LIN {X 0,Y 488.681,Z 523.609,A -85,B 0,C 180,E1 -6353.868,E2 -6353.868} C_VEL
LIN {X 0,Y 488.74,Z 523.606,A -85,B 0,C 180,E1 -6356.877,E2 -6356.877} C_VEL
LIN {X 0,Y 488.729,Z 523.605,A -85,B 0,C 180,E1 -6359.78,E2 -6359.78} C_VEL
LIN {X 0,Y 488.797,Z 523.6,A -85,B 0,C 180,E1 -6363.056,E2 -6363.056} C_VEL
LIN {X 0,Y 488.688,Z 523.606,A -85,B 0,C 180,E1 -6366.254,E2 -6366.254} C_VEL
LIN {X 0,Y 488.769,Z 523.791,A -85,B 0,C 180,E1 -6368.6,E2 -6368.6} C_VEL
LIN {X 0,Y 489.922,Z 530.451,A -85,B 0,C 180,E1 -6370.08,E2 -6370.08} C_VEL
LIN {X 0,Y 489.464,Z 545.093,A -85,B 0,C 180,E1 -6373.096,E2 -6373.096} C_VEL
LIN {X 0,Y 489.361,Z 548.713,A -85,B 0,C 180,E1 -6373.771,E2 -6373.771} C_VEL
LIN {X 0,Y 491.805,Z 562.137,A -85,B 0,C 180,E1 -6374.082,E2 -6374.082} C_VEL
LIN {X 0,Y 491.211,Z 655.586,A -85,B 0,C 180,E1 -6375.473,E2 -6375.473} C_VEL
LIN {X 0,Y 490.919,Z 668.738,A -85,B 0,C 180,E1 -6375.834,E2 -6375.834} C_VEL
LIN {X 0,Y 490.606,Z 680.814,A -85,B 0,C 180,E1 -6376.327,E2 -6376.327} C_VEL
LIN {X 0,Y 490.275,Z 691.758,A -85,B 0,C 180,E1 -6376.924,E2 -6376.924} C_VEL
LIN {X 0,Y 489.93,Z 702.578,A -85,B 0,C 180,E1 -6377.679,E2 -6377.679} C_VEL
LIN {X 0,Y 489.463,Z 713.275,A -85,B 0,C 180,E1 -6378.613,E2 -6378.613} C_VEL
LIN {X 0,Y 489.087,Z 722.892,A -85,B 0,C 180,E1 -6379.652,E2 -6379.652} C_VEL
LIN {X 0,Y 488.737,Z 730.772,A -85,B 0,C 180,E1 -6380.689,E2 -6380.689} C_VEL
LIN {X 0,Y 488.455,Z 738.473,A -85,B 0,C 180,E1 -6381.935,E2 -6381.935} C_VEL
LIN {X 0,Y 488.183,Z 745.539,A -85,B 0,C 180,E1 -6383.386,E2 -6383.386} C_VEL
LIN {X 0,Y 488.073,Z 750.246,A -85,B 0,C 180,E1 -6384.629,E2 -6384.629} C_VEL
LIN {X 0,Y 488.068,Z 753.846,A -85,B 0,C 180,E1 -6385.871,E2 -6385.871} C_VEL
LIN {X 0,Y 487.979,Z 755.709,A -85,B 0,C 180,E1 -6386.697,E2 -6386.697} C_VEL
LIN {X 0,Y 487.933,Z 757.116,A -85,B 0,C 180,E1 -6387.523,E2 -6387.523} C_VEL
LIN {X 0,Y 487.834,Z 758.735,A -85,B 0,C 180,E1 -6389.174,E2 -6389.174} C_VEL
LIN {X 0,Y 487.819,Z 758.973,A -85,B 0,C 180,E1 -6389.999,E2 -6389.999} C_VEL
LIN {X 0,Y 487.834,Z 758.789,A -85,B 0,C 180,E1 -6390.825,E2 -6390.825} C_VEL
LIN {X 0,Y 487.933,Z 757.242,A -85,B 0,C 180,E1 -6392.476,E2 -6392.476} C_VEL
LIN {X 0,Y 487.979,Z 755.889,A -85,B 0,C 180,E1 -6393.302,E2 -6393.302} C_VEL
LIN {X 0,Y 488.012,Z 753.026,A -85,B 0,C 180,E1 -6394.542,E2 -6394.542} C_VEL
LIN {X 0,Y 488.204,Z 748.083,A -85,B 0,C 180,E1 -6396.069,E2 -6396.069} C_VEL
LIN {X 0,Y 488.28,Z 742.168,A -85,B 0,C 180,E1 -6397.442,E2 -6397.442} C_VEL
LIN {X 0,Y 488.598,Z 735.386,A -85,B 0,C 180,E1 -6398.686,E2 -6398.686} C_VEL
LIN {X 0,Y 488.907,Z 726.92,A -85,B 0,C 180,E1 -6399.932,E2 -6399.932} C_VEL
LIN {X 0,Y 489.272,Z 718.209,A -85,B 0,C 180,E1 -6400.971,E2 -6400.971} C_VEL
LIN {X 0,Y 489.748,Z 707.478,A -85,B 0,C 180,E1 -6402.009,E2 -6402.009} C_VEL
LIN {X 0,Y 490.074,Z 696.27,A -85,B 0,C 180,E1 -6402.873,E2 -6402.873} C_VEL
LIN {X 0,Y 490.496,Z 684.645,A -85,B 0,C 180,E1 -6403.569,E2 -6403.569} C_VEL
LIN {X 0,Y 490.899,Z 671.996,A -85,B 0,C 180,E1 -6404.138,E2 -6404.138} C_VEL
LIN {X 0,Y 491.147,Z 659.517,A -85,B 0,C 180,E1 -6404.528,E2 -6404.528} C_VEL
LIN {X 0,Y 491.348,Z 643.583,A -85,B 0,C 180,E1 -6404.813,E2 -6404.813} C_VEL
LIN {X 0,Y 491.714,Z 561.306,A -85,B 0,C 180,E1 -6406.023,E2 -6406.023} C_VEL
LIN {X 0,Y 489.374,Z 548.902,A -85,B 0,C 180,E1 -6406.31,E2 -6406.31} C_VEL
LIN {X 0,Y 489.362,Z 547.534,A -85,B 0,C 180,E1 -6406.498,E2 -6406.498} C_VEL
LIN {X 0,Y 489.893,Z 531.929,A -85,B 0,C 180,E1 -6409.701,E2 -6409.701} C_VEL
LIN {X 0,Y 489.546,Z 527.949,A -85,B 0,C 180,E1 -6410.555,E2 -6410.555} C_VEL
LIN {X 0,Y 488.755,Z 523.632,A -85,B 0,C 180,E1 -6411.565,E2 -6411.565} C_VEL
LIN {X 0,Y 488.746,Z 523.607,A -85,B 0,C 180,E1 -6415.052,E2 -6415.052} C_VEL
LIN {X 0,Y 488.746,Z 523.608,A -85,B 0,C 180,E1 -6417.396,E2 -6417.396} C_VEL
LIN {X 0,Y 488.709,Z 523.603,A -85,B 0,C 180,E1 -6420.362,E2 -6420.362} C_VEL
LIN {X 0,Y 488.734,Z 523.608,A -85,B 0,C 180,E1 -6423.484,E2 -6423.484} C_VEL
LIN {X 0,Y 488.687,Z 523.606,A -85,B 0,C 180,E1 -6426.355,E2 -6426.355} C_VEL
LIN {X 0,Y 488.699,Z 523.611,A -85,B 0,C 180,E1 -6429.253,E2 -6429.253} C_VEL
LIN {X 0,Y 488.721,Z 523.61,A -85,B 0,C 180,E1 -6431.601,E2 -6431.601} C_VEL
LIN {X 0,Y 488.708,Z 523.601,A -85,B 0,C 180,E1 -6434.8,E2 -6434.8} C_VEL
LIN {X 0,Y 488.687,Z 523.616,A -85,B 0,C 180,E1 -6437.474,E2 -6437.474} C_VEL
LIN {X 0,Y 488.744,Z 523.595,A -85,B 0,C 180,E1 -6440.75,E2 -6440.75} C_VEL
LIN {X 0,Y 488.681,Z 523.611,A -85,B 0,C 180,E1 -6443.868,E2 -6443.868} C_VEL
LIN {X 0,Y 488.734,Z 523.603,A -85,B 0,C 180,E1 -6446.877,E2 -6446.877} C_VEL
LIN {X 0,Y 488.728,Z 523.607,A -85,B 0,C 180,E1 -6449.781,E2 -6449.781} C_VEL
LIN {X 0,Y 488.793,Z 523.593,A -85,B 0,C 180,E1 -6453.054,E2 -6453.054} C_VEL
LIN {X 0,Y 488.687,Z 523.606,A -85,B 0,C 180,E1 -6456.254,E2 -6456.254} C_VEL
LIN {X 0,Y 488.739,Z 523.602,A -85,B 0,C 180,E1 -6459.175,E2 -6459.175} C_VEL
LIN {X 0,Y 488.752,Z 523.604,A -85,B 0,C 180,E1 -6461.627,E2 -6461.627} C_VEL
LIN {X 0,Y 488.754,Z 523.597,A -85,B 0,C 180,E1 -6464.999,E2 -6464.999} C_VEL
LIN {X 0,Y 488.798,Z 523.592,A -85,B 0,C 180,E1 -6468.387,E2 -6468.387} C_VEL
LIN {X 0,Y 488.811,Z 523.597,A -85,B 0,C 180,E1 -6471.733,E2 -6471.733} C_VEL
LIN {X 0,Y 488.849,Z 523.588,A -85,B 0,C 180,E1 -6474.224,E2 -6474.224} C_VEL
LIN {X 0,Y 488.954,Z 523.576,A -85,B 0,C 180,E1 -6477.529,E2 -6477.529} C_VEL
LIN {X 0,Y 488.962,Z 523.576,A -85,B 0,C 180,E1 -6480,E2 -6480} C_VEL
LIN {X 0,Y 488.955,Z 523.571,A -85,B 0,C 180,E1 -6482.471,E2 -6482.471} C_VEL
LIN {X 0,Y 488.848,Z 523.593,A -85,B 0,C 180,E1 -6485.776,E2 -6485.776} C_VEL
LIN {X 0,Y 488.81,Z 523.591,A -85,B 0,C 180,E1 -6488.267,E2 -6488.267} C_VEL
LIN {X 0,Y 488.822,Z 523.596,A -85,B 0,C 180,E1 -6491.612,E2 -6491.612} C_VEL
LIN {X 0,Y 488.754,Z 523.599,A -85,B 0,C 180,E1 -6495.001,E2 -6495.001} C_VEL
LIN {X 0,Y 488.747,Z 523.6,A -85,B 0,C 180,E1 -6498.442,E2 -6498.442} C_VEL
LIN {X 0,Y 488.7,Z 523.606,A -85,B 0,C 180,E1 -6501.071,E2 -6501.071} C_VEL
LIN {X 0,Y 488.687,Z 523.615,A -85,B 0,C 180,E1 -6503.746,E2 -6503.746} C_VEL
LIN {X 0,Y 488.792,Z 523.592,A -85,B 0,C 180,E1 -6506.946,E2 -6506.946} C_VEL
LIN {X 0,Y 488.703,Z 523.604,A -85,B 0,C 180,E1 -6510.364,E2 -6510.364} C_VEL
LIN {X 0,Y 488.73,Z 523.609,A -85,B 0,C 180,E1 -6513.485,E2 -6513.485} C_VEL
LIN {X 0,Y 488.683,Z 523.599,A -85,B 0,C 180,E1 -6516.356,E2 -6516.356} C_VEL
LIN {X 0,Y 488.696,Z 523.609,A -85,B 0,C 180,E1 -6519.255,E2 -6519.255} C_VEL
LIN {X 0,Y 488.704,Z 523.609,A -85,B 0,C 180,E1 -6521.601,E2 -6521.601} C_VEL
LIN {X 0,Y 488.707,Z 523.606,A -85,B 0,C 180,E1 -6524.802,E2 -6524.802} C_VEL
LIN {X 0,Y 488.728,Z 523.604,A -85,B 0,C 180,E1 -6527.48,E2 -6527.48} C_VEL
LIN {X 0,Y 488.739,Z 523.598,A -85,B 0,C 180,E1 -6530.751,E2 -6530.751} C_VEL
LIN {X 0,Y 488.681,Z 523.613,A -85,B 0,C 180,E1 -6533.869,E2 -6533.869} C_VEL
LIN {X 0,Y 488.737,Z 523.596,A -85,B 0,C 180,E1 -6536.878,E2 -6536.878} C_VEL
LIN {X 0,Y 488.722,Z 523.579,A -85,B 0,C 180,E1 -6539.782,E2 -6539.782} C_VEL
LIN {X 0,Y 488.791,Z 523.587,A -85,B 0,C 180,E1 -6543.057,E2 -6543.057} C_VEL
LIN {X 0,Y 488.791,Z 523.664,A -85,B 0,C 180,E1 -6544.812,E2 -6544.812} C_VEL
LIN {X 0,Y 489.553,Z 527.685,A -85,B 0,C 180,E1 -6545.624,E2 -6545.624} C_VEL
LIN {X 0,Y 490.749,Z 534.364,A -85,B 0,C 180,E1 -6546.859,E2 -6546.859} C_VEL
LIN {X 0,Y 490.077,Z 551.858,A -85,B 0,C 180,E1 -6549.869,E2 -6549.869} C_VEL
LIN {X 0,Y 489.463,Z 569.569,A -85,B 0,C 180,E1 -6552.882,E2 -6552.882} C_VEL
LIN {X 0,Y 489.365,Z 574.51,A -85,B 0,C 180,E1 -6553.695,E2 -6553.695} C_VEL
LIN {X 0,Y 490.061,Z 579.414,A -85,B 0,C 180,E1 -6553.83,E2 -6553.83} C_VEL
LIN {X 0,Y 491.733,Z 590.249,A -85,B 0,C 180,E1 -6554.047,E2 -6554.047} C_VEL
LIN {X 0,Y 491.141,Z 682.718,A -85,B 0,C 180,E1 -6555.419,E2 -6555.419} C_VEL
LIN {X 0,Y 490.851,Z 695.983,A -85,B 0,C 180,E1 -6555.781,E2 -6555.781} C_VEL
LIN {X 0,Y 490.517,Z 708.151,A -85,B 0,C 180,E1 -6556.273,E2 -6556.273} C_VEL
LIN {X 0,Y 490.094,Z 720.568,A -85,B 0,C 180,E1 -6556.956,E2 -6556.956} C_VEL
LIN {X 0,Y 489.627,Z 732.037,A -85,B 0,C 180,E1 -6557.778,E2 -6557.778} C_VEL
LIN {X 0,Y 489.256,Z 742.483,A -85,B 0,C 180,E1 -6558.714,E2 -6558.714} C_VEL
LIN {X 0,Y 488.874,Z 751.025,A -85,B 0,C 180,E1 -6559.649,E2 -6559.649} C_VEL
LIN {X 0,Y 488.593,Z 758.906,A -85,B 0,C 180,E1 -6560.688,E2 -6560.688} C_VEL
LIN {X 0,Y 488.327,Z 766.606,A -85,B 0,C 180,E1 -6561.934,E2 -6561.934} C_VEL
LIN {X 0,Y 488.1,Z 773.701,A -85,B 0,C 180,E1 -6563.386,E2 -6563.386} C_VEL
LIN {X 0,Y 488.033,Z 778.425,A -85,B 0,C 180,E1 -6564.63,E2 -6564.63} C_VEL
LIN {X 0,Y 487.934,Z 782.035,A -85,B 0,C 180,E1 -6565.871,E2 -6565.871} C_VEL
LIN {X 0,Y 487.965,Z 783.899,A -85,B 0,C 180,E1 -6566.698,E2 -6566.698} C_VEL
LIN {X 0,Y 487.89,Z 786.286,A -85,B 0,C 180,E1 -6568.35,E2 -6568.35} C_VEL
LIN {X 0,Y 487.819,Z 787.107,A -85,B 0,C 180,E1 -6570.001,E2 -6570.001} C_VEL
LIN {X 0,Y 487.89,Z 786.283,A -85,B 0,C 180,E1 -6571.652,E2 -6571.652} C_VEL
LIN {X 0,Y 487.965,Z 783.892,A -85,B 0,C 180,E1 -6573.303,E2 -6573.303} C_VEL
LIN {X 0,Y 487.928,Z 780.957,A -85,B 0,C 180,E1 -6574.544,E2 -6574.544} C_VEL
LIN {X 0,Y 488.06,Z 776.989,A -85,B 0,C 180,E1 -6575.786,E2 -6575.786} C_VEL
LIN {X 0,Y 488.184,Z 770.876,A -85,B 0,C 180,E1 -6577.237,E2 -6577.237} C_VEL
LIN {X 0,Y 488.382,Z 764.198,A -85,B 0,C 180,E1 -6578.483,E2 -6578.483} C_VEL
LIN {X 0,Y 488.702,Z 755.914,A -85,B 0,C 180,E1 -6579.729,E2 -6579.729} C_VEL
LIN {X 0,Y 489.013,Z 747.424,A -85,B 0,C 180,E1 -6580.769,E2 -6580.769} C_VEL
LIN {X 0,Y 489.508,Z 736.936,A -85,B 0,C 180,E1 -6581.806,E2 -6581.806} C_VEL
LIN {X 0,Y 489.842,Z 725.58,A -85,B 0,C 180,E1 -6582.711,E2 -6582.711} C_VEL
LIN {X 0,Y 490.288,Z 713.26,A -85,B 0,C 180,E1 -6583.471,E2 -6583.471} C_VEL
LIN {X 0,Y 490.725,Z 700.919,A -85,B 0,C 180,E1 -6584.039,E2 -6584.039} C_VEL
LIN {X 0,Y 491.05,Z 688.242,A -85,B 0,C 180,E1 -6584.453,E2 -6584.453} C_VEL
LIN {X 0,Y 491.266,Z 675.001,A -85,B 0,C 180,E1 -6584.711,E2 -6584.711} C_VEL
LIN {X 0,Y 491.59,Z 588.729,A -85,B 0,C 180,E1 -6585.98,E2 -6585.98} C_VEL
LIN {X 0,Y 489.357,Z 574.659,A -85,B 0,C 180,E1 -6586.292,E2 -6586.292} C_VEL
LIN {X 0,Y 489.946,Z 556.914,A -85,B 0,C 180,E1 -6589.265,E2 -6589.265} C_VEL
LIN {X 0,Y 490.637,Z 537.874,A -85,B 0,C 180,E1 -6592.531,E2 -6592.531} C_VEL
LIN {X 0,Y 490.755,Z 534.35,A -85,B 0,C 180,E1 -6593.143,E2 -6593.143} C_VEL
LIN {X 0,Y 488.834,Z 523.999,A -85,B 0,C 180,E1 -6595.075,E2 -6595.075} C_VEL
LIN {X 0,Y 488.776,Z 523.603,A -85,B 0,C 180,E1 -6595.263,E2 -6595.263} C_VEL
LIN {X 0,Y 488.75,Z 523.605,A -85,B 0,C 180,E1 -6597.397,E2 -6597.397} C_VEL
LIN {X 0,Y 488.714,Z 523.608,A -85,B 0,C 180,E1 -6600.363,E2 -6600.363} C_VEL
LIN {X 0,Y 488.738,Z 523.603,A -85,B 0,C 180,E1 -6603.484,E2 -6603.484} C_VEL
LIN {X 0,Y 488.686,Z 523.614,A -85,B 0,C 180,E1 -6606.355,E2 -6606.355} C_VEL
LIN {X 0,Y 488.704,Z 523.607,A -85,B 0,C 180,E1 -6609.254,E2 -6609.254} C_VEL
LIN {X 0,Y 488.711,Z 523.608,A -85,B 0,C 180,E1 -6611.6,E2 -6611.6} C_VEL
LIN {X 0,Y 488.705,Z 523.609,A -85,B 0,C 180,E1 -6614.803,E2 -6614.803} C_VEL
LIN {X 0,Y 488.695,Z 523.609,A -85,B 0,C 180,E1 -6617.475,E2 -6617.475} C_VEL
LIN {X 0,Y 488.736,Z 523.604,A -85,B 0,C 180,E1 -6619.677,E2 -6619.677} C_VEL
LIN {X 0,Y 488.685,Z 523.612,A -85,B 0,C 180,E1 -6622.841,E2 -6622.841} C_VEL
LIN {X 0,Y 488.737,Z 523.608,A -85,B 0,C 180,E1 -6625.888,E2 -6625.888} C_VEL
LIN {X 0,Y 488.695,Z 523.612,A -85,B 0,C 180,E1 -6628.82,E2 -6628.82} C_VEL
LIN {X 0,Y 488.749,Z 523.607,A -85,B 0,C 180,E1 -6631.671,E2 -6631.671} C_VEL
LIN {X 0,Y 488.801,Z 523.734,A -85,B 0,C 180,E1 -6633.789,E2 -6633.789} C_VEL
LIN {X 0,Y 490.59,Z 533.223,A -85,B 0,C 180,E1 -6635.248,E2 -6635.248} C_VEL
LIN {X 0,Y 490.416,Z 548.756,A -85,B 0,C 180,E1 -6637.459,E2 -6637.459} C_VEL
LIN {X 0,Y 490.098,Z 565.541,A -85,B 0,C 180,E1 -6639.869,E2 -6639.869} C_VEL
LIN {X 0,Y 489.634,Z 584.967,A -85,B 0,C 180,E1 -6642.672,E2 -6642.672} C_VEL
LIN {X 0,Y 489.216,Z 605.451,A -85,B 0,C 180,E1 -6645.652,E2 -6645.652} C_VEL
LIN {X 0,Y 489.02,Z 616.715,A -85,B 0,C 180,E1 -6647.261,E2 -6647.261} C_VEL
LIN {X 0,Y 490.209,Z 627.69,A -85,B 0,C 180,E1 -6647.486,E2 -6647.486} C_VEL
LIN {X 0,Y 489.863,Z 696.03,A -85,B 0,C 180,E1 -6648.57,E2 -6648.57} C_VEL
LIN {X 0,Y 489.666,Z 706.138,A -85,B 0,C 180,E1 -6648.854,E2 -6648.854} C_VEL
LIN {X 0,Y 489.473,Z 715.662,A -85,B 0,C 180,E1 -6649.242,E2 -6649.242} C_VEL
LIN {X 0,Y 489.269,Z 725.188,A -85,B 0,C 180,E1 -6649.761,E2 -6649.761} C_VEL
LIN {X 0,Y 488.981,Z 735.411,A -85,B 0,C 180,E1 -6650.486,E2 -6650.486} C_VEL
LIN {X 0,Y 488.71,Z 744.347,A -85,B 0,C 180,E1 -6651.315,E2 -6651.315} C_VEL
LIN {X 0,Y 488.521,Z 749.955,A -85,B 0,C 180,E1 -6651.937,E2 -6651.937} C_VEL
LIN {X 0,Y 488.36,Z 756.343,A -85,B 0,C 180,E1 -6652.787,E2 -6652.787} C_VEL
LIN {X 0,Y 488.28,Z 761.064,A -85,B 0,C 180,E1 -6653.534,E2 -6653.534} C_VEL
LIN {X 0,Y 488.182,Z 764.784,A -85,B 0,C 180,E1 -6654.216,E2 -6654.216} C_VEL
LIN {X 0,Y 488.013,Z 768.529,A -85,B 0,C 180,E1 -6655.043,E2 -6655.043} C_VEL
LIN {X 0,Y 488.024,Z 772.817,A -85,B 0,C 180,E1 -6656.284,E2 -6656.284} C_VEL
LIN {X 0,Y 487.912,Z 775.791,A -85,B 0,C 180,E1 -6657.523,E2 -6657.523} C_VEL
LIN {X 0,Y 487.89,Z 777.114,A -85,B 0,C 180,E1 -6658.349,E2 -6658.349} C_VEL
LIN {X 0,Y 487.832,Z 777.944,A -85,B 0,C 180,E1 -6659.175,E2 -6659.175} C_VEL
LIN {X 0,Y 487.817,Z 778.248,A -85,B 0,C 180,E1 -6660,E2 -6660} C_VEL
LIN {X 0,Y 487.833,Z 777.976,A -85,B 0,C 180,E1 -6660.826,E2 -6660.826} C_VEL
LIN {X 0,Y 487.891,Z 777.213,A -85,B 0,C 180,E1 -6661.651,E2 -6661.651} C_VEL
LIN {X 0,Y 487.913,Z 775.959,A -85,B 0,C 180,E1 -6662.477,E2 -6662.477} C_VEL
LIN {X 0,Y 488.024,Z 773.058,A -85,B 0,C 180,E1 -6663.716,E2 -6663.716} C_VEL
LIN {X 0,Y 488.002,Z 768.887,A -85,B 0,C 180,E1 -6664.957,E2 -6664.957} C_VEL
LIN {X 0,Y 488.253,Z 763.064,A -85,B 0,C 180,E1 -6666.198,E2 -6666.198} C_VEL
LIN {X 0,Y 488.327,Z 756.977,A -85,B 0,C 180,E1 -6667.214,E2 -6667.214} C_VEL
LIN {X 0,Y 488.518,Z 750.724,A -85,B 0,C 180,E1 -6668.063,E2 -6668.063} C_VEL
LIN {X 0,Y 488.784,Z 742.329,A -85,B 0,C 180,E1 -6668.996,E2 -6668.996} C_VEL
LIN {X 0,Y 489.105,Z 732.681,A -85,B 0,C 180,E1 -6669.825,E2 -6669.825} C_VEL
LIN {X 0,Y 489.364,Z 723.46,A -85,B 0,C 180,E1 -6670.446,E2 -6670.446} C_VEL
LIN {X 0,Y 489.547,Z 714.618,A -85,B 0,C 180,E1 -6670.913,E2 -6670.913} C_VEL
LIN {X 0,Y 489.68,Z 704.075,A -85,B 0,C 180,E1 -6671.329,E2 -6671.329} C_VEL
LIN {X 0,Y 489.903,Z 691.2,A -85,B 0,C 180,E1 -6671.634,E2 -6671.634} C_VEL
LIN {X 0,Y 490.139,Z 625.929,A -85,B 0,C 180,E1 -6672.645,E2 -6672.645} C_VEL
LIN {X 0,Y 489,Z 616.477,A -85,B 0,C 180,E1 -6672.848,E2 -6672.848} C_VEL
LIN {X 0,Y 489.468,Z 596.198,A -85,B 0,C 180,E1 -6675.841,E2 -6675.841} C_VEL
LIN {X 0,Y 490.088,Z 573.271,A -85,B 0,C 180,E1 -6679.258,E2 -6679.258} C_VEL
LIN {X 0,Y 490.633,Z 552.885,A -85,B 0,C 180,E1 -6682.309,E2 -6682.309} C_VEL
LIN {X 0,Y 491.09,Z 536.633,A -85,B 0,C 180,E1 -6684.746,E2 -6684.746} C_VEL
LIN {X 0,Y 489.915,Z 529.365,A -85,B 0,C 180,E1 -6685.901,E2 -6685.901} C_VEL
LIN {X 0,Y 488.806,Z 523.674,A -85,B 0,C 180,E1 -6686.858,E2 -6686.858} C_VEL
LIN {X 0,Y 488.727,Z 523.608,A -85,B 0,C 180,E1 -6690.219,E2 -6690.219} C_VEL
LIN {X 0,Y 488.739,Z 523.609,A -85,B 0,C 180,E1 -6693.484,E2 -6693.484} C_VEL
LIN {X 0,Y 488.688,Z 523.609,A -85,B 0,C 180,E1 -6696.355,E2 -6696.355} C_VEL
LIN {X 0,Y 488.705,Z 523.609,A -85,B 0,C 180,E1 -6699.254,E2 -6699.254} C_VEL
LIN {X 0,Y 488.71,Z 523.59,A -85,B 0,C 180,E1 -6701.6,E2 -6701.6} C_VEL
LIN {X 0,Y 488.705,Z 523.602,A -85,B 0,C 180,E1 -6704.803,E2 -6704.803} C_VEL
LIN {X 0,Y 488.688,Z 523.608,A -85,B 0,C 180,E1 -6707.694,E2 -6707.694} C_VEL
LIN {X 0,Y 488.025,Z 523.689,A -85,B 0,C 180,E1 -6708.383,E2 -6708.383} C_VEL
LIN {X 0,Y 485.195,Z 524.033,A -85,B 0,C 180,E1 -6709.501,E2 -6709.501} C_VEL
LIN {X 0,Y 482.794,Z 524.332,A -85,B 0,C 180,E1 -6710.403,E2 -6710.403} C_VEL
LIN {X 0,Y 481.751,Z 524.463,A -85,B 0,C 180,E1 -6711.099,E2 -6711.099} C_VEL
LIN {X 0,Y 481.66,Z 524.475,A -85,B 0,C 180,E1 -6711.334,E2 -6711.334} C_VEL
LIN {X 0,Y 481.664,Z 524.487,A -85,B 0,C 180,E1 -6714.796,E2 -6714.796} C_VEL
LIN {X 0,Y 481.661,Z 524.484,A -85,B 0,C 180,E1 -6717.811,E2 -6717.811} C_VEL
LIN {X 0,Y 481.705,Z 524.482,A -85,B 0,C 180,E1 -6721.218,E2 -6721.218} C_VEL
LIN {X 0,Y 481.701,Z 524.481,A -85,B 0,C 180,E1 -6724.042,E2 -6724.042} C_VEL
LIN {X 0,Y 481.679,Z 524.486,A -85,B 0,C 180,E1 -6726.812,E2 -6726.812} C_VEL
LIN {X 0,Y 481.697,Z 524.571,A -85,B 0,C 180,E1 -6728.382,E2 -6728.382} C_VEL
LIN {X 0,Y 482.973,Z 531.668,A -85,B 0,C 180,E1 -6730.003,E2 -6730.003} C_VEL
LIN {X 0,Y 482.458,Z 546.33,A -85,B 0,C 180,E1 -6733.061,E2 -6733.061} C_VEL
LIN {X 0,Y 482.397,Z 548.784,A -85,B 0,C 180,E1 -6733.519,E2 -6733.519} C_VEL
LIN {X 0,Y 483.572,Z 554.995,A -85,B 0,C 180,E1 -6733.691,E2 -6733.691} C_VEL
LIN {X 0,Y 484.986,Z 563.576,A -85,B 0,C 180,E1 -6733.87,E2 -6733.87} C_VEL
LIN {X 0,Y 484.363,Z 655.818,A -85,B 0,C 180,E1 -6735.263,E2 -6735.263} C_VEL
LIN {X 0,Y 484.068,Z 668.96,A -85,B 0,C 180,E1 -6735.63,E2 -6735.63} C_VEL
LIN {X 0,Y 483.731,Z 681.032,A -85,B 0,C 180,E1 -6736.129,E2 -6736.129} C_VEL
LIN {X 0,Y 483.362,Z 692.174,A -85,B 0,C 180,E1 -6736.746,E2 -6736.746} C_VEL
LIN {X 0,Y 483.002,Z 702.791,A -85,B 0,C 180,E1 -6737.499,E2 -6737.499} C_VEL
LIN {X 0,Y 482.522,Z 713.486,A -85,B 0,C 180,E1 -6738.447,E2 -6738.447} C_VEL
LIN {X 0,Y 482.099,Z 723.102,A -85,B 0,C 180,E1 -6739.5,E2 -6739.5} C_VEL
LIN {X 0,Y 481.72,Z 730.981,A -85,B 0,C 180,E1 -6740.553,E2 -6740.553} C_VEL
LIN {X 0,Y 481.406,Z 738.682,A -85,B 0,C 180,E1 -6741.816,E2 -6741.816} C_VEL
LIN {X 0,Y 481.12,Z 745.747,A -85,B 0,C 180,E1 -6743.288,E2 -6743.288} C_VEL
LIN {X 0,Y 481.021,Z 750.453,A -85,B 0,C 180,E1 -6744.55,E2 -6744.55} C_VEL
LIN {X 0,Y 480.968,Z 754.052,A -85,B 0,C 180,E1 -6745.809,E2 -6745.809} C_VEL
LIN {X 0,Y 480.91,Z 755.915,A -85,B 0,C 180,E1 -6746.648,E2 -6746.648} C_VEL
LIN {X 0,Y 480.846,Z 757.321,A -85,B 0,C 180,E1 -6747.486,E2 -6747.486} C_VEL
LIN {X 0,Y 480.823,Z 758.321,A -85,B 0,C 180,E1 -6748.324,E2 -6748.324} C_VEL
LIN {X 0,Y 480.743,Z 759.177,A -85,B 0,C 180,E1 -6749.999,E2 -6749.999} C_VEL
LIN {X 0,Y 480.76,Z 758.992,A -85,B 0,C 180,E1 -6750.837,E2 -6750.837} C_VEL
LIN {X 0,Y 480.824,Z 758.409,A -85,B 0,C 180,E1 -6751.674,E2 -6751.674} C_VEL
LIN {X 0,Y 480.91,Z 756.092,A -85,B 0,C 180,E1 -6753.35,E2 -6753.35} C_VEL
LIN {X 0,Y 480.915,Z 753.23,A -85,B 0,C 180,E1 -6754.609,E2 -6754.609} C_VEL
LIN {X 0,Y 481.128,Z 749.342,A -85,B 0,C 180,E1 -6755.868,E2 -6755.868} C_VEL
LIN {X 0,Y 481.192,Z 744.338,A -85,B 0,C 180,E1 -6757.131,E2 -6757.131} C_VEL
LIN {X 0,Y 481.45,Z 738.035,A -85,B 0,C 180,E1 -6758.393,E2 -6758.393} C_VEL
LIN {X 0,Y 481.776,Z 730.14,A -85,B 0,C 180,E1 -6759.657,E2 -6759.657} C_VEL
LIN {X 0,Y 482.101,Z 722.094,A -85,B 0,C 180,E1 -6760.711,E2 -6760.711} C_VEL
LIN {X 0,Y 482.606,Z 712.268,A -85,B 0,C 180,E1 -6761.763,E2 -6761.763} C_VEL
LIN {X 0,Y 483.016,Z 702.609,A -85,B 0,C 180,E1 -6762.606,E2 -6762.606} C_VEL
LIN {X 0,Y 483.327,Z 691.991,A -85,B 0,C 180,E1 -6763.356,E2 -6763.356} C_VEL
LIN {X 0,Y 483.804,Z 679.565,A -85,B 0,C 180,E1 -6764.028,E2 -6764.028} C_VEL
LIN {X 0,Y 484.148,Z 666.208,A -85,B 0,C 180,E1 -6764.554,E2 -6764.554} C_VEL
LIN {X 0,Y 484.392,Z 653.697,A -85,B 0,C 180,E1 -6764.869,E2 -6764.869} C_VEL
LIN {X 0,Y 484.917,Z 562.268,A -85,B 0,C 180,E1 -6766.242,E2 -6766.242} C_VEL
LIN {X 0,Y 482.477,Z 549.323,A -85,B 0,C 180,E1 -6766.539,E2 -6766.539} C_VEL
LIN {X 0,Y 482.382,Z 548.273,A -85,B 0,C 180,E1 -6766.646,E2 -6766.646} C_VEL
LIN {X 0,Y 482.945,Z 533.134,A -85,B 0,C 180,E1 -6769.775,E2 -6769.775} C_VEL
LIN {X 0,Y 482.467,Z 528.525,A -85,B 0,C 180,E1 -6770.783,E2 -6770.783} C_VEL
LIN {X 0,Y 481.701,Z 524.532,A -85,B 0,C 180,E1 -6771.728,E2 -6771.728} C_VEL
LIN {X 0,Y 481.712,Z 524.481,A -85,B 0,C 180,E1 -6775.236,E2 -6775.236} C_VEL
LIN {X 0,Y 481.7,Z 524.481,A -85,B 0,C 180,E1 -6777.831,E2 -6777.831} C_VEL
LIN {X 0,Y 481.646,Z 524.484,A -85,B 0,C 180,E1 -6780.71,E2 -6780.71} C_VEL
LIN {X 0,Y 481.695,Z 524.484,A -85,B 0,C 180,E1 -6783.732,E2 -6783.732} C_VEL
LIN {X 0,Y 481.627,Z 524.486,A -85,B 0,C 180,E1 -6786.746,E2 -6786.746} C_VEL
LIN {X 0,Y 481.674,Z 524.48,A -85,B 0,C 180,E1 -6789.939,E2 -6789.939} C_VEL
LIN {X 0,Y 481.663,Z 524.489,A -85,B 0,C 180,E1 -6793.296,E2 -6793.296} C_VEL
LIN {X 0,Y 481.654,Z 524.486,A -85,B 0,C 180,E1 -6795.64,E2 -6795.64} C_VEL
LIN {X 0,Y 481.663,Z 524.485,A -85,B 0,C 180,E1 -6798.959,E2 -6798.959} C_VEL
LIN {X 0,Y 481.698,Z 524.475,A -85,B 0,C 180,E1 -6801.143,E2 -6801.143} C_VEL
LIN {X 0,Y 481.664,Z 524.483,A -85,B 0,C 180,E1 -6804.794,E2 -6804.794} C_VEL
LIN {X 0,Y 481.668,Z 524.487,A -85,B 0,C 180,E1 -6807.325,E2 -6807.325} C_VEL
LIN {X 0,Y 481.682,Z 524.48,A -85,B 0,C 180,E1 -6810.259,E2 -6810.259} C_VEL
LIN {X 0,Y 481.746,Z 524.471,A -85,B 0,C 180,E1 -6813.112,E2 -6813.112} C_VEL
LIN {X 0,Y 481.671,Z 524.483,A -85,B 0,C 180,E1 -6815.886,E2 -6815.886} C_VEL
LIN {X 0,Y 481.695,Z 524.477,A -85,B 0,C 180,E1 -6819.027,E2 -6819.027} C_VEL
LIN {X 0,Y 481.7,Z 524.476,A -85,B 0,C 180,E1 -6822.158,E2 -6822.158} C_VEL
LIN {X 0,Y 481.735,Z 524.47,A -85,B 0,C 180,E1 -6824.775,E2 -6824.775} C_VEL
LIN {X 0,Y 481.743,Z 524.471,A -85,B 0,C 180,E1 -6828.215,E2 -6828.215} C_VEL
LIN {X 0,Y 481.756,Z 524.476,A -85,B 0,C 180,E1 -6831.612,E2 -6831.612} C_VEL
LIN {X 0,Y 481.81,Z 524.465,A -85,B 0,C 180,E1 -6834.139,E2 -6834.139} C_VEL
LIN {X 0,Y 481.921,Z 524.451,A -85,B 0,C 180,E1 -6837.492,E2 -6837.492} C_VEL
LIN {X 0,Y 481.933,Z 524.452,A -85,B 0,C 180,E1 -6840,E2 -6840} C_VEL
LIN {X 0,Y 481.922,Z 524.447,A -85,B 0,C 180,E1 -6842.507,E2 -6842.507} C_VEL
LIN {X 0,Y 481.809,Z 524.469,A -85,B 0,C 180,E1 -6845.86,E2 -6845.86} C_VEL
LIN {X 0,Y 481.755,Z 524.469,A -85,B 0,C 180,E1 -6848.388,E2 -6848.388} C_VEL
LIN {X 0,Y 481.787,Z 524.472,A -85,B 0,C 180,E1 -6851.784,E2 -6851.784} C_VEL
LIN {X 0,Y 481.735,Z 524.476,A -85,B 0,C 180,E1 -6855.224,E2 -6855.224} C_VEL
LIN {X 0,Y 481.705,Z 524.477,A -85,B 0,C 180,E1 -6858.722,E2 -6858.722} C_VEL
LIN {X 0,Y 481.64,Z 524.489,A -85,B 0,C 180,E1 -6861.395,E2 -6861.395} C_VEL
LIN {X 0,Y 481.671,Z 524.484,A -85,B 0,C 180,E1 -6864.114,E2 -6864.114} C_VEL
LIN {X 0,Y 481.745,Z 524.471,A -85,B 0,C 180,E1 -6867.141,E2 -6867.141} C_VEL
LIN {X 0,Y 481.672,Z 524.487,A -85,B 0,C 180,E1 -6869.742,E2 -6869.742} C_VEL
LIN {X 0,Y 481.667,Z 524.482,A -85,B 0,C 180,E1 -6872.675,E2 -6872.675} C_VEL
LIN {X 0,Y 481.637,Z 524.483,A -85,B 0,C 180,E1 -6875.71,E2 -6875.71} C_VEL
LIN {X 0,Y 481.666,Z 524.482,A -85,B 0,C 180,E1 -6878.86,E2 -6878.86} C_VEL
LIN {X 0,Y 481.648,Z 524.483,A -85,B 0,C 180,E1 -6881.914,E2 -6881.914} C_VEL
LIN {X 0,Y 481.655,Z 524.484,A -85,B 0,C 180,E1 -6884.458,E2 -6884.458} C_VEL
LIN {X 0,Y 481.685,Z 524.477,A -85,B 0,C 180,E1 -6886.847,E2 -6886.847} C_VEL
LIN {X 0,Y 481.686,Z 524.48,A -85,B 0,C 180,E1 -6890.062,E2 -6890.062} C_VEL
LIN {X 0,Y 481.625,Z 524.482,A -85,B 0,C 180,E1 -6893.254,E2 -6893.254} C_VEL
LIN {X 0,Y 481.707,Z 524.472,A -85,B 0,C 180,E1 -6896.331,E2 -6896.331} C_VEL
LIN {X 0,Y 481.649,Z 524.453,A -85,B 0,C 180,E1 -6899.418,E2 -6899.418} C_VEL
LIN {X 0,Y 481.699,Z 524.48,A -85,B 0,C 180,E1 -6902.169,E2 -6902.169} C_VEL
LIN {X 0,Y 481.767,Z 524.629,A -85,B 0,C 180,E1 -6904.649,E2 -6904.649} C_VEL
LIN {X 0,Y 483.692,Z 534.902,A -85,B 0,C 180,E1 -6906.629,E2 -6906.629} C_VEL
LIN {X 0,Y 483.482,Z 543.914,A -85,B 0,C 180,E1 -6908.218,E2 -6908.218} C_VEL
LIN {X 0,Y 482.785,Z 561.808,A -85,B 0,C 180,E1 -6911.322,E2 -6911.322} C_VEL
LIN {X 0,Y 482.409,Z 574.501,A -85,B 0,C 180,E1 -6913.469,E2 -6913.469} C_VEL
LIN {X 0,Y 484.913,Z 591.467,A -85,B 0,C 180,E1 -6913.838,E2 -6913.838} C_VEL
LIN {X 0,Y 484.288,Z 682.514,A -85,B 0,C 180,E1 -6915.208,E2 -6915.208} C_VEL
LIN {X 0,Y 483.968,Z 695.779,A -85,B 0,C 180,E1 -6915.574,E2 -6915.574} C_VEL
LIN {X 0,Y 483.621,Z 707.946,A -85,B 0,C 180,E1 -6916.074,E2 -6916.074} C_VEL
LIN {X 0,Y 483.176,Z 720.235,A -85,B 0,C 180,E1 -6916.758,E2 -6916.758} C_VEL
LIN {X 0,Y 482.664,Z 731.831,A -85,B 0,C 180,E1 -6917.599,E2 -6917.599} C_VEL
LIN {X 0,Y 482.236,Z 742.276,A -85,B 0,C 180,E1 -6918.548,E2 -6918.548} C_VEL
LIN {X 0,Y 481.867,Z 750.819,A -85,B 0,C 180,E1 -6919.496,E2 -6919.496} C_VEL
LIN {X 0,Y 481.543,Z 758.7,A -85,B 0,C 180,E1 -6920.551,E2 -6920.551} C_VEL
LIN {X 0,Y 481.257,Z 766.4,A -85,B 0,C 180,E1 -6921.815,E2 -6921.815} C_VEL
LIN {X 0,Y 481.019,Z 773.496,A -85,B 0,C 180,E1 -6923.288,E2 -6923.288} C_VEL
LIN {X 0,Y 480.949,Z 778.219,A -85,B 0,C 180,E1 -6924.55,E2 -6924.55} C_VEL
LIN {X 0,Y 480.834,Z 781.83,A -85,B 0,C 180,E1 -6925.81,E2 -6925.81} C_VEL
LIN {X 0,Y 480.889,Z 783.694,A -85,B 0,C 180,E1 -6926.649,E2 -6926.649} C_VEL
LIN {X 0,Y 480.792,Z 786.082,A -85,B 0,C 180,E1 -6928.325,E2 -6928.325} C_VEL
LIN {X 0,Y 480.743,Z 786.903,A -85,B 0,C 180,E1 -6930.001,E2 -6930.001} C_VEL
LIN {X 0,Y 480.76,Z 786.686,A -85,B 0,C 180,E1 -6930.838,E2 -6930.838} C_VEL
LIN {X 0,Y 480.823,Z 785.083,A -85,B 0,C 180,E1 -6932.514,E2 -6932.514} C_VEL
LIN {X 0,Y 480.89,Z 783.688,A -85,B 0,C 180,E1 -6933.352,E2 -6933.352} C_VEL
LIN {X 0,Y 480.845,Z 780.753,A -85,B 0,C 180,E1 -6934.612,E2 -6934.612} C_VEL
LIN {X 0,Y 480.962,Z 776.783,A -85,B 0,C 180,E1 -6935.872,E2 -6935.872} C_VEL
LIN {X 0,Y 481.113,Z 770.67,A -85,B 0,C 180,E1 -6937.344,E2 -6937.344} C_VEL
LIN {X 0,Y 481.341,Z 763.993,A -85,B 0,C 180,E1 -6938.608,E2 -6938.608} C_VEL
LIN {X 0,Y 481.677,Z 755.709,A -85,B 0,C 180,E1 -6939.872,E2 -6939.872} C_VEL
LIN {X 0,Y 482.026,Z 747.219,A -85,B 0,C 180,E1 -6940.927,E2 -6940.927} C_VEL
LIN {X 0,Y 482.535,Z 736.731,A -85,B 0,C 180,E1 -6941.979,E2 -6941.979} C_VEL
LIN {X 0,Y 482.883,Z 725.4,A -85,B 0,C 180,E1 -6942.895,E2 -6942.895} C_VEL
LIN {X 0,Y 483.388,Z 713.055,A -85,B 0,C 180,E1 -6943.666,E2 -6943.666} C_VEL
LIN {X 0,Y 483.821,Z 700.714,A -85,B 0,C 180,E1 -6944.244,E2 -6944.244} C_VEL
LIN {X 0,Y 484.182,Z 688.038,A -85,B 0,C 180,E1 -6944.662,E2 -6944.662} C_VEL
LIN {X 0,Y 484.396,Z 674.796,A -85,B 0,C 180,E1 -6944.924,E2 -6944.924} C_VEL
LIN {X 0,Y 484.809,Z 589.878,A -85,B 0,C 180,E1 -6946.189,E2 -6946.189} C_VEL
LIN {X 0,Y 482.407,Z 574.706,A -85,B 0,C 180,E1 -6946.517,E2 -6946.517} C_VEL
LIN {X 0,Y 482.437,Z 570.622,A -85,B 0,C 180,E1 -6947.158,E2 -6947.158} C_VEL
LIN {X 0,Y 483.063,Z 554.202,A -85,B 0,C 180,E1 -6949.993,E2 -6949.993} C_VEL
LIN {X 0,Y 483.803,Z 536.428,A -85,B 0,C 180,E1 -6953.093,E2 -6953.093} C_VEL
LIN {X 0,Y 482.322,Z 527.489,A -85,B 0,C 180,E1 -6954.767,E2 -6954.767} C_VEL
LIN {X 0,Y 481.771,Z 524.622,A -85,B 0,C 180,E1 -6955.352,E2 -6955.352} C_VEL
LIN {X 0,Y 481.704,Z 524.477,A -85,B 0,C 180,E1 -6957.832,E2 -6957.832} C_VEL
LIN {X 0,Y 481.65,Z 524.489,A -85,B 0,C 180,E1 -6960.711,E2 -6960.711} C_VEL
LIN {X 0,Y 481.701,Z 524.481,A -85,B 0,C 180,E1 -6963.733,E2 -6963.733} C_VEL
LIN {X 0,Y 481.629,Z 524.49,A -85,B 0,C 180,E1 -6966.747,E2 -6966.747} C_VEL
LIN {X 0,Y 481.68,Z 524.486,A -85,B 0,C 180,E1 -6969.941,E2 -6969.941} C_VEL
LIN {X 0,Y 481.642,Z 524.487,A -85,B 0,C 180,E1 -6973.3,E2 -6973.3} C_VEL
LIN {X 0,Y 481.657,Z 524.487,A -85,B 0,C 180,E1 -6975.642,E2 -6975.642} C_VEL
LIN {X 0,Y 481.66,Z 524.485,A -85,B 0,C 180,E1 -6978.958,E2 -6978.958} C_VEL
LIN {X 0,Y 481.659,Z 524.49,A -85,B 0,C 180,E1 -6981.993,E2 -6981.993} C_VEL
LIN {X 0,Y 481.696,Z 524.481,A -85,B 0,C 180,E1 -6985.318,E2 -6985.318} C_VEL
LIN {X 0,Y 481.648,Z 524.492,A -85,B 0,C 180,E1 -6988.312,E2 -6988.312} C_VEL
LIN {X 0,Y 481.704,Z 524.482,A -85,B 0,C 180,E1 -6991.219,E2 -6991.219} C_VEL
LIN {X 0,Y 481.776,Z 524.713,A -85,B 0,C 180,E1 -6993.625,E2 -6993.625} C_VEL
LIN {X 0,Y 483.768,Z 535.734,A -85,B 0,C 180,E1 -6995.312,E2 -6995.312} C_VEL
LIN {X 0,Y 483.384,Z 554.492,A -85,B 0,C 180,E1 -6998.005,E2 -6998.005} C_VEL
LIN {X 0,Y 482.921,Z 573.838,A -85,B 0,C 180,E1 -7000.828,E2 -7000.828} C_VEL
LIN {X 0,Y 482.46,Z 595.838,A -85,B 0,C 180,E1 -7004.035,E2 -7004.035} C_VEL
LIN {X 0,Y 481.998,Z 616.689,A -85,B 0,C 180,E1 -7007.064,E2 -7007.064} C_VEL
LIN {X 0,Y 483.284,Z 628.154,A -85,B 0,C 180,E1 -7007.309,E2 -7007.309} C_VEL
LIN {X 0,Y 482.875,Z 696.43,A -85,B 0,C 180,E1 -7008.429,E2 -7008.429} C_VEL
LIN {X 0,Y 482.681,Z 706.399,A -85,B 0,C 180,E1 -7008.717,E2 -7008.717} C_VEL
LIN {X 0,Y 482.473,Z 716.404,A -85,B 0,C 180,E1 -7009.137,E2 -7009.137} C_VEL
LIN {X 0,Y 482.235,Z 726.65,A -85,B 0,C 180,E1 -7009.716,E2 -7009.716} C_VEL
LIN {X 0,Y 481.922,Z 736.426,A -85,B 0,C 180,E1 -7010.451,E2 -7010.451} C_VEL
LIN {X 0,Y 481.7,Z 744.226,A -85,B 0,C 180,E1 -7011.188,E2 -7011.188} C_VEL
LIN {X 0,Y 481.425,Z 751.524,A -85,B 0,C 180,E1 -7012.028,E2 -7012.028} C_VEL
LIN {X 0,Y 481.264,Z 757.813,A -85,B 0,C 180,E1 -7012.912,E2 -7012.912} C_VEL
LIN {X 0,Y 481.2,Z 763.231,A -85,B 0,C 180,E1 -7013.841,E2 -7013.841} C_VEL
LIN {X 0,Y 480.947,Z 768.535,A -85,B 0,C 180,E1 -7014.97,E2 -7014.97} C_VEL
LIN {X 0,Y 480.949,Z 772.846,A -85,B 0,C 180,E1 -7016.23,E2 -7016.23} C_VEL
LIN {X 0,Y 480.827,Z 775.832,A -85,B 0,C 180,E1 -7017.487,E2 -7017.487} C_VEL
LIN {X 0,Y 480.791,Z 777.163,A -85,B 0,C 180,E1 -7018.325,E2 -7018.325} C_VEL
LIN {X 0,Y 480.758,Z 777.998,A -85,B 0,C 180,E1 -7019.162,E2 -7019.162} C_VEL
LIN {X 0,Y 480.741,Z 778.302,A -85,B 0,C 180,E1 -7020,E2 -7020} C_VEL
LIN {X 0,Y 480.759,Z 778.028,A -85,B 0,C 180,E1 -7020.838,E2 -7020.838} C_VEL
LIN {X 0,Y 480.793,Z 777.261,A -85,B 0,C 180,E1 -7021.675,E2 -7021.675} C_VEL
LIN {X 0,Y 480.828,Z 775.999,A -85,B 0,C 180,E1 -7022.513,E2 -7022.513} C_VEL
LIN {X 0,Y 480.948,Z 773.085,A -85,B 0,C 180,E1 -7023.77,E2 -7023.77} C_VEL
LIN {X 0,Y 480.937,Z 768.891,A -85,B 0,C 180,E1 -7025.03,E2 -7025.03} C_VEL
LIN {X 0,Y 481.173,Z 763.833,A -85,B 0,C 180,E1 -7026.143,E2 -7026.143} C_VEL
LIN {X 0,Y 481.248,Z 758.169,A -85,B 0,C 180,E1 -7027.131,E2 -7027.131} C_VEL
LIN {X 0,Y 481.422,Z 752.295,A -85,B 0,C 180,E1 -7027.972,E2 -7027.972} C_VEL
LIN {X 0,Y 481.659,Z 745.17,A -85,B 0,C 180,E1 -7028.813,E2 -7028.813} C_VEL
LIN {X 0,Y 481.92,Z 737.588,A -85,B 0,C 180,E1 -7029.549,E2 -7029.549} C_VEL
LIN {X 0,Y 482.217,Z 728.23,A -85,B 0,C 180,E1 -7030.285,E2 -7030.285} C_VEL
LIN {X 0,Y 482.471,Z 717.575,A -85,B 0,C 180,E1 -7030.916,E2 -7030.916} C_VEL
LIN {X 0,Y 482.676,Z 707.971,A -85,B 0,C 180,E1 -7031.336,E2 -7031.336} C_VEL
LIN {X 0,Y 482.796,Z 698.709,A -85,B 0,C 180,E1 -7031.626,E2 -7031.626} C_VEL
LIN {X 0,Y 482.975,Z 685.813,A -85,B 0,C 180,E1 -7031.872,E2 -7031.872} C_VEL
LIN {X 0,Y 483.207,Z 626.513,A -85,B 0,C 180,E1 -7032.816,E2 -7032.816} C_VEL
LIN {X 0,Y 482.002,Z 616.449,A -85,B 0,C 180,E1 -7033.038,E2 -7033.038} C_VEL
LIN {X 0,Y 482.482,Z 596.134,A -85,B 0,C 180,E1 -7036.067,E2 -7036.067} C_VEL
LIN {X 0,Y 483.106,Z 574.21,A -85,B 0,C 180,E1 -7039.363,E2 -7039.363} C_VEL
LIN {X 0,Y 483.685,Z 553.958,A -85,B 0,C 180,E1 -7042.422,E2 -7042.422} C_VEL
LIN {X 0,Y 484.158,Z 537.61,A -85,B 0,C 180,E1 -7044.895,E2 -7044.895} C_VEL
LIN {X 0,Y 482.537,Z 528.442,A -85,B 0,C 180,E1 -7046.374,E2 -7046.374} C_VEL
LIN {X 0,Y 481.762,Z 524.545,A -85,B 0,C 180,E1 -7047.053,E2 -7047.053} C_VEL
LIN {X 0,Y 481.682,Z 524.488,A -85,B 0,C 180,E1 -7049.741,E2 -7049.741} C_VEL
LIN {X 0,Y 481.676,Z 524.483,A -85,B 0,C 180,E1 -7052.674,E2 -7052.674} C_VEL
LIN {X 0,Y 481.642,Z 524.493,A -85,B 0,C 180,E1 -7055.709,E2 -7055.709} C_VEL
LIN {X 0,Y 481.675,Z 524.481,A -85,B 0,C 180,E1 -7058.859,E2 -7058.859} C_VEL
LIN {X 0,Y 481.655,Z 524.465,A -85,B 0,C 180,E1 -7061.913,E2 -7061.913} C_VEL
LIN {X 0,Y 481.658,Z 524.478,A -85,B 0,C 180,E1 -7064.458,E2 -7064.458} C_VEL
LIN {X 0,Y 481.652,Z 524.483,A -85,B 0,C 180,E1 -7067.839,E2 -7067.839} C_VEL
LIN {X 0,Y 481.663,Z 524.469,A -85,B 0,C 180,E1 -7070.654,E2 -7070.654} C_VEL
LIN {X 0,Y 481.66,Z 524.475,A -85,B 0,C 180,E1 -7071.334,E2 -7071.334} C_VEL
LIN {X 0,Y 480.979,Z 524.567,A -85,B 0,C 180,E1 -7072.032,E2 -7072.032} C_VEL
LIN {X 0,Y 478.134,Z 524.929,A -85,B 0,C 180,E1 -7073.166,E2 -7073.166} C_VEL
LIN {X 0,Y 475.734,Z 525.228,A -85,B 0,C 180,E1 -7074.08,E2 -7074.08} C_VEL
LIN {X 0,Y 474.698,Z 525.355,A -85,B 0,C 180,E1 -7074.786,E2 -7074.786} C_VEL
LIN {X 0,Y 474.61,Z 525.362,A -85,B 0,C 180,E1 -7075.025,E2 -7075.025} C_VEL
LIN {X 0,Y 474.639,Z 525.359,A -85,B 0,C 180,E1 -7077.787,E2 -7077.787} C_VEL
LIN {X 0,Y 474.629,Z 525.365,A -85,B 0,C 180,E1 -7080.884,E2 -7080.884} C_VEL
LIN {X 0,Y 474.663,Z 525.358,A -85,B 0,C 180,E1 -7083.628,E2 -7083.628} C_VEL
LIN {X 0,Y 474.64,Z 525.36,A -85,B 0,C 180,E1 -7086.641,E2 -7086.641} C_VEL
LIN {X 0,Y 474.683,Z 525.556,A -85,B 0,C 180,E1 -7088.246,E2 -7088.246} C_VEL
LIN {X 0,Y 476.013,Z 532.887,A -85,B 0,C 180,E1 -7089.923,E2 -7089.923} C_VEL
LIN {X 0,Y 475.519,Z 546.523,A -85,B 0,C 180,E1 -7092.806,E2 -7092.806} C_VEL
LIN {X 0,Y 475.465,Z 549.1,A -85,B 0,C 180,E1 -7093.282,E2 -7093.282} C_VEL
LIN {X 0,Y 478.195,Z 564.162,A -85,B 0,C 180,E1 -7093.64,E2 -7093.64} C_VEL
LIN {X 0,Y 477.514,Z 656.046,A -85,B 0,C 180,E1 -7095.047,E2 -7095.047} C_VEL
LIN {X 0,Y 477.215,Z 669.18,A -85,B 0,C 180,E1 -7095.419,E2 -7095.419} C_VEL
LIN {X 0,Y 476.85,Z 681.248,A -85,B 0,C 180,E1 -7095.925,E2 -7095.925} C_VEL
LIN {X 0,Y 476.452,Z 692.626,A -85,B 0,C 180,E1 -7096.566,E2 -7096.566} C_VEL
LIN {X 0,Y 476.018,Z 704.29,A -85,B 0,C 180,E1 -7097.421,E2 -7097.421} C_VEL
LIN {X 0,Y 475.51,Z 714.762,A -85,B 0,C 180,E1 -7098.382,E2 -7098.382} C_VEL
LIN {X 0,Y 475.092,Z 723.313,A -85,B 0,C 180,E1 -7099.343,E2 -7099.343} C_VEL
LIN {X 0,Y 474.723,Z 731.19,A -85,B 0,C 180,E1 -7100.412,E2 -7100.412} C_VEL
LIN {X 0,Y 474.371,Z 738.89,A -85,B 0,C 180,E1 -7101.694,E2 -7101.694} C_VEL
LIN {X 0,Y 474.069,Z 745.955,A -85,B 0,C 180,E1 -7103.188,E2 -7103.188} C_VEL
LIN {X 0,Y 473.972,Z 750.659,A -85,B 0,C 180,E1 -7104.468,E2 -7104.468} C_VEL
LIN {X 0,Y 473.869,Z 754.259,A -85,B 0,C 180,E1 -7105.747,E2 -7105.747} C_VEL
LIN {X 0,Y 473.842,Z 756.12,A -85,B 0,C 180,E1 -7106.598,E2 -7106.598} C_VEL
LIN {X 0,Y 473.763,Z 757.527,A -85,B 0,C 180,E1 -7107.449,E2 -7107.449} C_VEL
LIN {X 0,Y 473.689,Z 759.144,A -85,B 0,C 180,E1 -7109.149,E2 -7109.149} C_VEL
LIN {X 0,Y 473.67,Z 759.381,A -85,B 0,C 180,E1 -7109.999,E2 -7109.999} C_VEL
LIN {X 0,Y 473.689,Z 759.196,A -85,B 0,C 180,E1 -7110.849,E2 -7110.849} C_VEL
LIN {X 0,Y 473.763,Z 757.65,A -85,B 0,C 180,E1 -7112.55,E2 -7112.55} C_VEL
LIN {X 0,Y 473.841,Z 756.295,A -85,B 0,C 180,E1 -7113.4,E2 -7113.4} C_VEL
LIN {X 0,Y 473.826,Z 753.433,A -85,B 0,C 180,E1 -7114.679,E2 -7114.679} C_VEL
LIN {X 0,Y 474.071,Z 749.545,A -85,B 0,C 180,E1 -7115.956,E2 -7115.956} C_VEL
LIN {X 0,Y 474.142,Z 744.54,A -85,B 0,C 180,E1 -7117.237,E2 -7117.237} C_VEL
LIN {X 0,Y 474.421,Z 738.237,A -85,B 0,C 180,E1 -7118.518,E2 -7118.518} C_VEL
LIN {X 0,Y 474.759,Z 730.341,A -85,B 0,C 180,E1 -7119.801,E2 -7119.801} C_VEL
LIN {X 0,Y 475.127,Z 722.294,A -85,B 0,C 180,E1 -7120.87,E2 -7120.87} C_VEL
LIN {X 0,Y 475.655,Z 712.467,A -85,B 0,C 180,E1 -7121.937,E2 -7121.937} C_VEL
LIN {X 0,Y 476.081,Z 702.806,A -85,B 0,C 180,E1 -7122.792,E2 -7122.792} C_VEL
LIN {X 0,Y 476.416,Z 692.431,A -85,B 0,C 180,E1 -7123.538,E2 -7123.538} C_VEL
LIN {X 0,Y 476.922,Z 679.758,A -85,B 0,C 180,E1 -7124.235,E2 -7124.235} C_VEL
LIN {X 0,Y 477.297,Z 666.396,A -85,B 0,C 180,E1 -7124.768,E2 -7124.768} C_VEL
LIN {X 0,Y 477.547,Z 653.871,A -85,B 0,C 180,E1 -7125.087,E2 -7125.087} C_VEL
LIN {X 0,Y 478.022,Z 562.552,A -85,B 0,C 180,E1 -7126.481,E2 -7126.481} C_VEL
LIN {X 0,Y 475.481,Z 549.431,A -85,B 0,C 180,E1 -7126.793,E2 -7126.793} C_VEL
LIN {X 0,Y 475.415,Z 548.464,A -85,B 0,C 180,E1 -7126.897,E2 -7126.897} C_VEL
LIN {X 0,Y 476.028,Z 533.297,A -85,B 0,C 180,E1 -7130.075,E2 -7130.075} C_VEL
LIN {X 0,Y 474.649,Z 525.387,A -85,B 0,C 180,E1 -7131.925,E2 -7131.925} C_VEL
LIN {X 0,Y 474.67,Z 525.356,A -85,B 0,C 180,E1 -7135.427,E2 -7135.427} C_VEL
LIN {X 0,Y 474.645,Z 525.357,A -85,B 0,C 180,E1 -7138.281,E2 -7138.281} C_VEL
LIN {X 0,Y 474.599,Z 525.367,A -85,B 0,C 180,E1 -7141.216,E2 -7141.216} C_VEL
LIN {X 0,Y 474.632,Z 525.36,A -85,B 0,C 180,E1 -7144.24,E2 -7144.24} C_VEL
LIN {X 0,Y 474.59,Z 525.37,A -85,B 0,C 180,E1 -7147.383,E2 -7147.383} C_VEL
LIN {X 0,Y 474.625,Z 525.36,A -85,B 0,C 180,E1 -7149.647,E2 -7149.647} C_VEL
LIN {X 0,Y 474.632,Z 525.361,A -85,B 0,C 180,E1 -7152.931,E2 -7152.931} C_VEL
LIN {X 0,Y 474.605,Z 525.363,A -85,B 0,C 180,E1 -7155.894,E2 -7155.894} C_VEL
LIN {X 0,Y 474.636,Z 525.361,A -85,B 0,C 180,E1 -7159.038,E2 -7159.038} C_VEL
LIN {X 0,Y 474.615,Z 525.356,A -85,B 0,C 180,E1 -7161.702,E2 -7161.702} C_VEL
LIN {X 0,Y 474.625,Z 525.36,A -85,B 0,C 180,E1 -7164.726,E2 -7164.726} C_VEL
LIN {X 0,Y 474.632,Z 525.361,A -85,B 0,C 180,E1 -7167.787,E2 -7167.787} C_VEL
LIN {X 0,Y 474.626,Z 525.36,A -85,B 0,C 180,E1 -7170.882,E2 -7170.882} C_VEL
LIN {X 0,Y 474.661,Z 525.361,A -85,B 0,C 180,E1 -7173.628,E2 -7173.628} C_VEL
LIN {X 0,Y 474.629,Z 525.357,A -85,B 0,C 180,E1 -7176.641,E2 -7176.641} C_VEL
LIN {X 0,Y 474.65,Z 525.357,A -85,B 0,C 180,E1 -7180.089,E2 -7180.089} C_VEL
LIN {X 0,Y 474.644,Z 525.355,A -85,B 0,C 180,E1 -7182.774,E2 -7182.774} C_VEL
LIN {X 0,Y 474.641,Z 525.36,A -85,B 0,C 180,E1 -7185.421,E2 -7185.421} C_VEL
LIN {X 0,Y 474.696,Z 525.35,A -85,B 0,C 180,E1 -7188.037,E2 -7188.037} C_VEL
LIN {X 0,Y 474.721,Z 525.349,A -85,B 0,C 180,E1 -7191.486,E2 -7191.486} C_VEL
LIN {X 0,Y 474.772,Z 525.342,A -85,B 0,C 180,E1 -7194.052,E2 -7194.052} C_VEL
LIN {X 0,Y 474.887,Z 525.326,A -85,B 0,C 180,E1 -7197.455,E2 -7197.455} C_VEL
LIN {X 0,Y 474.869,Z 525.329,A -85,B 0,C 180,E1 -7200.848,E2 -7200.848} C_VEL
LIN {X 0,Y 474.888,Z 525.323,A -85,B 0,C 180,E1 -7202.545,E2 -7202.545} C_VEL
LIN {X 0,Y 474.772,Z 525.344,A -85,B 0,C 180,E1 -7205.948,E2 -7205.948} C_VEL
LIN {X 0,Y 474.72,Z 525.345,A -85,B 0,C 180,E1 -7208.514,E2 -7208.514} C_VEL
LIN {X 0,Y 474.731,Z 525.349,A -85,B 0,C 180,E1 -7211.962,E2 -7211.962} C_VEL
LIN {X 0,Y 474.673,Z 525.354,A -85,B 0,C 180,E1 -7215.768,E2 -7215.768} C_VEL
LIN {X 0,Y 474.658,Z 525.356,A -85,B 0,C 180,E1 -7219.011,E2 -7219.011} C_VEL
LIN {X 0,Y 474.584,Z 525.367,A -85,B 0,C 180,E1 -7221.729,E2 -7221.729} C_VEL
LIN {X 0,Y 474.652,Z 525.356,A -85,B 0,C 180,E1 -7224.493,E2 -7224.493} C_VEL
LIN {X 0,Y 474.692,Z 525.351,A -85,B 0,C 180,E1 -7227.339,E2 -7227.339} C_VEL
LIN {X 0,Y 474.599,Z 525.361,A -85,B 0,C 180,E1 -7230.811,E2 -7230.811} C_VEL
LIN {X 0,Y 474.632,Z 525.36,A -85,B 0,C 180,E1 -7233.985,E2 -7233.985} C_VEL
LIN {X 0,Y 474.569,Z 525.356,A -85,B 0,C 180,E1 -7236.901,E2 -7236.901} C_VEL
LIN {X 0,Y 474.623,Z 525.368,A -85,B 0,C 180,E1 -7239.648,E2 -7239.648} C_VEL
LIN {X 0,Y 474.61,Z 525.355,A -85,B 0,C 180,E1 -7242.935,E2 -7242.935} C_VEL
LIN {X 0,Y 474.614,Z 525.363,A -85,B 0,C 180,E1 -7245.897,E2 -7245.897} C_VEL
LIN {X 0,Y 474.642,Z 525.359,A -85,B 0,C 180,E1 -7249.039,E2 -7249.039} C_VEL
LIN {X 0,Y 474.613,Z 525.353,A -85,B 0,C 180,E1 -7251.704,E2 -7251.704} C_VEL
LIN {X 0,Y 474.626,Z 525.361,A -85,B 0,C 180,E1 -7254.727,E2 -7254.727} C_VEL
LIN {X 0,Y 474.635,Z 525.332,A -85,B 0,C 180,E1 -7257.789,E2 -7257.789} C_VEL
LIN {X 0,Y 474.623,Z 525.36,A -85,B 0,C 180,E1 -7260.885,E2 -7260.885} C_VEL
LIN {X 0,Y 474.661,Z 525.337,A -85,B 0,C 180,E1 -7263.629,E2 -7263.629} C_VEL
LIN {X 0,Y 474.689,Z 525.459,A -85,B 0,C 180,E1 -7264.416,E2 -7264.416} C_VEL
LIN {X 0,Y 475.8,Z 531.159,A -85,B 0,C 180,E1 -7265.571,E2 -7265.571} C_VEL
LIN {X 0,Y 476.842,Z 537.538,A -85,B 0,C 180,E1 -7266.781,E2 -7266.781} C_VEL
LIN {X 0,Y 476.12,Z 554.029,A -85,B 0,C 180,E1 -7269.704,E2 -7269.704} C_VEL
LIN {X 0,Y 475.477,Z 570.443,A -85,B 0,C 180,E1 -7272.585,E2 -7272.585} C_VEL
LIN {X 0,Y 475.412,Z 574.307,A -85,B 0,C 180,E1 -7273.219,E2 -7273.219} C_VEL
LIN {X 0,Y 478.083,Z 592.265,A -85,B 0,C 180,E1 -7273.616,E2 -7273.616} C_VEL
LIN {X 0,Y 477.431,Z 682.314,A -85,B 0,C 180,E1 -7274.991,E2 -7274.991} C_VEL
LIN {X 0,Y 477.105,Z 695.577,A -85,B 0,C 180,E1 -7275.362,E2 -7275.362} C_VEL
LIN {X 0,Y 476.725,Z 707.743,A -85,B 0,C 180,E1 -7275.868,E2 -7275.868} C_VEL
LIN {X 0,Y 476.25,Z 720.031,A -85,B 0,C 180,E1 -7276.561,E2 -7276.561} C_VEL
LIN {X 0,Y 475.698,Z 731.717,A -85,B 0,C 180,E1 -7277.422,E2 -7277.422} C_VEL
LIN {X 0,Y 475.27,Z 742.071,A -85,B 0,C 180,E1 -7278.377,E2 -7278.377} C_VEL
LIN {X 0,Y 474.853,Z 750.614,A -85,B 0,C 180,E1 -7279.339,E2 -7279.339} C_VEL
LIN {X 0,Y 474.498,Z 758.494,A -85,B 0,C 180,E1 -7280.409,E2 -7280.409} C_VEL
LIN {X 0,Y 474.184,Z 766.194,A -85,B 0,C 180,E1 -7281.692,E2 -7281.692} C_VEL
LIN {X 0,Y 473.936,Z 773.29,A -85,B 0,C 180,E1 -7283.188,E2 -7283.188} C_VEL
LIN {X 0,Y 473.865,Z 778.014,A -85,B 0,C 180,E1 -7284.469,E2 -7284.469} C_VEL
LIN {X 0,Y 473.74,Z 781.625,A -85,B 0,C 180,E1 -7285.747,E2 -7285.747} C_VEL
LIN {X 0,Y 473.797,Z 783.489,A -85,B 0,C 180,E1 -7286.599,E2 -7286.599} C_VEL
LIN {X 0,Y 473.741,Z 784.883,A -85,B 0,C 180,E1 -7287.45,E2 -7287.45} C_VEL
LIN {X 0,Y 473.688,Z 786.484,A -85,B 0,C 180,E1 -7289.151,E2 -7289.151} C_VEL
LIN {X 0,Y 473.669,Z 786.699,A -85,B 0,C 180,E1 -7290.001,E2 -7290.001} C_VEL
LIN {X 0,Y 473.688,Z 786.482,A -85,B 0,C 180,E1 -7290.851,E2 -7290.851} C_VEL
LIN {X 0,Y 473.741,Z 784.878,A -85,B 0,C 180,E1 -7292.552,E2 -7292.552} C_VEL
LIN {X 0,Y 473.797,Z 783.483,A -85,B 0,C 180,E1 -7293.402,E2 -7293.402} C_VEL
LIN {X 0,Y 473.768,Z 780.548,A -85,B 0,C 180,E1 -7294.681,E2 -7294.681} C_VEL
LIN {X 0,Y 473.868,Z 776.577,A -85,B 0,C 180,E1 -7295.96,E2 -7295.96} C_VEL
LIN {X 0,Y 474.033,Z 770.464,A -85,B 0,C 180,E1 -7297.455,E2 -7297.455} C_VEL
LIN {X 0,Y 474.302,Z 763.787,A -85,B 0,C 180,E1 -7298.737,E2 -7298.737} C_VEL
LIN {X 0,Y 474.627,Z 755.503,A -85,B 0,C 180,E1 -7300.02,E2 -7300.02} C_VEL
LIN {X 0,Y 475.03,Z 747.013,A -85,B 0,C 180,E1 -7301.09,E2 -7301.09} C_VEL
LIN {X 0,Y 475.562,Z 736.669,A -85,B 0,C 180,E1 -7302.144,E2 -7302.144} C_VEL
LIN {X 0,Y 475.944,Z 724.858,A -85,B 0,C 180,E1 -7303.112,E2 -7303.112} C_VEL
LIN {X 0,Y 476.485,Z 712.849,A -85,B 0,C 180,E1 -7303.868,E2 -7303.868} C_VEL
LIN {X 0,Y 476.948,Z 700.507,A -85,B 0,C 180,E1 -7304.453,E2 -7304.453} C_VEL
LIN {X 0,Y 477.309,Z 687.829,A -85,B 0,C 180,E1 -7304.878,E2 -7304.878} C_VEL
LIN {X 0,Y 477.545,Z 674.584,A -85,B 0,C 180,E1 -7305.143,E2 -7305.143} C_VEL
LIN {X 0,Y 477.97,Z 590.508,A -85,B 0,C 180,E1 -7306.414,E2 -7306.414} C_VEL
LIN {X 0,Y 475.424,Z 574.273,A -85,B 0,C 180,E1 -7306.783,E2 -7306.783} C_VEL
LIN {X 0,Y 475.972,Z 557.93,A -85,B 0,C 180,E1 -7309.606,E2 -7309.606} C_VEL
LIN {X 0,Y 476.763,Z 540.059,A -85,B 0,C 180,E1 -7312.766,E2 -7312.766} C_VEL
LIN {X 0,Y 476.751,Z 536.247,A -85,B 0,C 180,E1 -7313.455,E2 -7313.455} C_VEL
LIN {X 0,Y 474.711,Z 525.588,A -85,B 0,C 180,E1 -7315.532,E2 -7315.532} C_VEL
LIN {X 0,Y 474.666,Z 525.352,A -85,B 0,C 180,E1 -7316.372,E2 -7316.372} C_VEL
LIN {X 0,Y 474.625,Z 525.351,A -85,B 0,C 180,E1 -7319.252,E2 -7319.252} C_VEL
LIN {X 0,Y 474.619,Z 525.367,A -85,B 0,C 180,E1 -7322.431,E2 -7322.431} C_VEL
LIN {X 0,Y 474.618,Z 525.361,A -85,B 0,C 180,E1 -7325.469,E2 -7325.469} C_VEL
LIN {X 0,Y 474.615,Z 525.365,A -85,B 0,C 180,E1 -7328.458,E2 -7328.458} C_VEL
LIN {X 0,Y 474.631,Z 525.361,A -85,B 0,C 180,E1 -7330.959,E2 -7330.959} C_VEL
LIN {X 0,Y 474.61,Z 525.367,A -85,B 0,C 180,E1 -7334.105,E2 -7334.105} C_VEL
LIN {X 0,Y 474.618,Z 525.363,A -85,B 0,C 180,E1 -7337.066,E2 -7337.066} C_VEL
LIN {X 0,Y 474.648,Z 525.362,A -85,B 0,C 180,E1 -7340.454,E2 -7340.454} C_VEL
LIN {X 0,Y 474.595,Z 525.368,A -85,B 0,C 180,E1 -7343.677,E2 -7343.677} C_VEL
LIN {X 0,Y 474.646,Z 525.361,A -85,B 0,C 180,E1 -7346.78,E2 -7346.78} C_VEL
LIN {X 0,Y 474.609,Z 525.369,A -85,B 0,C 180,E1 -7349.77,E2 -7349.77} C_VEL
LIN {X 0,Y 474.729,Z 525.354,A -85,B 0,C 180,E1 -7353.158,E2 -7353.158} C_VEL
LIN {X 0,Y 474.767,Z 525.742,A -85,B 0,C 180,E1 -7353.427,E2 -7353.427} C_VEL
LIN {X 0,Y 476.85,Z 536.897,A -85,B 0,C 180,E1 -7355.163,E2 -7355.163} C_VEL
LIN {X 0,Y 476.465,Z 557.49,A -85,B 0,C 180,E1 -7358.156,E2 -7358.156} C_VEL
LIN {X 0,Y 475.893,Z 580.166,A -85,B 0,C 180,E1 -7361.487,E2 -7361.487} C_VEL
LIN {X 0,Y 475.332,Z 603.948,A -85,B 0,C 180,E1 -7365.004,E2 -7365.004} C_VEL
LIN {X 0,Y 475.003,Z 616.507,A -85,B 0,C 180,E1 -7366.848,E2 -7366.848} C_VEL
LIN {X 0,Y 475.741,Z 622.242,A -85,B 0,C 180,E1 -7367.002,E2 -7367.002} C_VEL
LIN {X 0,Y 476.361,Z 630.351,A -85,B 0,C 180,E1 -7367.159,E2 -7367.159} C_VEL
LIN {X 0,Y 475.895,Z 697.024,A -85,B 0,C 180,E1 -7368.284,E2 -7368.284} C_VEL
LIN {X 0,Y 475.7,Z 706.812,A -85,B 0,C 180,E1 -7368.576,E2 -7368.576} C_VEL
LIN {X 0,Y 475.499,Z 716.174,A -85,B 0,C 180,E1 -7368.976,E2 -7368.976} C_VEL
LIN {X 0,Y 475.258,Z 726.479,A -85,B 0,C 180,E1 -7369.563,E2 -7369.563} C_VEL
LIN {X 0,Y 474.935,Z 736.323,A -85,B 0,C 180,E1 -7370.31,E2 -7370.31} C_VEL
LIN {X 0,Y 474.686,Z 744.148,A -85,B 0,C 180,E1 -7371.057,E2 -7371.057} C_VEL
LIN {X 0,Y 474.375,Z 751.469,A -85,B 0,C 180,E1 -7371.909,E2 -7371.909} C_VEL
LIN {X 0,Y 474.216,Z 757.502,A -85,B 0,C 180,E1 -7372.763,E2 -7372.763} C_VEL
LIN {X 0,Y 474.126,Z 763.52,A -85,B 0,C 180,E1 -7373.805,E2 -7373.805} C_VEL
LIN {X 0,Y 473.885,Z 768.542,A -85,B 0,C 180,E1 -7374.895,E2 -7374.895} C_VEL
LIN {X 0,Y 473.874,Z 772.877,A -85,B 0,C 180,E1 -7376.173,E2 -7376.173} C_VEL
LIN {X 0,Y 473.746,Z 775.877,A -85,B 0,C 180,E1 -7377.449,E2 -7377.449} C_VEL
LIN {X 0,Y 473.697,Z 777.214,A -85,B 0,C 180,E1 -7378.3,E2 -7378.3} C_VEL
LIN {X 0,Y 473.686,Z 778.052,A -85,B 0,C 180,E1 -7379.15,E2 -7379.15} C_VEL
LIN {X 0,Y 473.668,Z 778.357,A -85,B 0,C 180,E1 -7380,E2 -7380} C_VEL
LIN {X 0,Y 473.687,Z 778.08,A -85,B 0,C 180,E1 -7380.85,E2 -7380.85} C_VEL
LIN {X 0,Y 473.699,Z 777.308,A -85,B 0,C 180,E1 -7381.7,E2 -7381.7} C_VEL
LIN {X 0,Y 473.747,Z 776.039,A -85,B 0,C 180,E1 -7382.551,E2 -7382.551} C_VEL
LIN {X 0,Y 473.872,Z 773.108,A -85,B 0,C 180,E1 -7383.827,E2 -7383.827} C_VEL
LIN {X 0,Y 473.875,Z 768.896,A -85,B 0,C 180,E1 -7385.105,E2 -7385.105} C_VEL
LIN {X 0,Y 474.099,Z 764.107,A -85,B 0,C 180,E1 -7386.179,E2 -7386.179} C_VEL
LIN {X 0,Y 474.183,Z 758.117,A -85,B 0,C 180,E1 -7387.237,E2 -7387.237} C_VEL
LIN {X 0,Y 474.372,Z 752.213,A -85,B 0,C 180,E1 -7388.091,E2 -7388.091} C_VEL
LIN {X 0,Y 474.621,Z 745.052,A -85,B 0,C 180,E1 -7388.945,E2 -7388.945} C_VEL
LIN {X 0,Y 474.922,Z 737.433,A -85,B 0,C 180,E1 -7389.691,E2 -7389.691} C_VEL
LIN {X 0,Y 475.223,Z 728.025,A -85,B 0,C 180,E1 -7390.438,E2 -7390.438} C_VEL
LIN {X 0,Y 475.497,Z 717.242,A -85,B 0,C 180,E1 -7391.078,E2 -7391.078} C_VEL
LIN {X 0,Y 475.719,Z 707.532,A -85,B 0,C 180,E1 -7391.504,E2 -7391.504} C_VEL
LIN {X 0,Y 475.847,Z 698.088,A -85,B 0,C 180,E1 -7391.798,E2 -7391.798} C_VEL
LIN {X 0,Y 476.069,Z 682.4,A -85,B 0,C 180,E1 -7392.086,E2 -7392.086} C_VEL
LIN {X 0,Y 476.263,Z 626.83,A -85,B 0,C 180,E1 -7392.993,E2 -7392.993} C_VEL
LIN {X 0,Y 475.041,Z 616.807,A -85,B 0,C 180,E1 -7393.208,E2 -7393.208} C_VEL
LIN {X 0,Y 475.201,Z 608.954,A -85,B 0,C 180,E1 -7394.343,E2 -7394.343} C_VEL
LIN {X 0,Y 475.642,Z 590.188,A -85,B 0,C 180,E1 -7397.189,E2 -7397.189} C_VEL
LIN {X 0,Y 476.259,Z 571.254,A -85,B 0,C 180,E1 -7400.066,E2 -7400.066} C_VEL
LIN {X 0,Y 476.822,Z 552.052,A -85,B 0,C 180,E1 -7402.991,E2 -7402.991} C_VEL
LIN {X 0,Y 477.203,Z 538.568,A -85,B 0,C 180,E1 -7405.051,E2 -7405.051} C_VEL
LIN {X 0,Y 474.737,Z 525.447,A -85,B 0,C 180,E1 -7407.23,E2 -7407.23} C_VEL
LIN {X 0,Y 474.608,Z 525.365,A -85,B 0,C 180,E1 -7410.81,E2 -7410.81} C_VEL
LIN {X 0,Y 474.642,Z 525.362,A -85,B 0,C 180,E1 -7413.984,E2 -7413.984} C_VEL
LIN {X 0,Y 474.576,Z 525.367,A -85,B 0,C 180,E1 -7416.899,E2 -7416.899} C_VEL
LIN {X 0,Y 474.631,Z 525.355,A -85,B 0,C 180,E1 -7419.647,E2 -7419.647} C_VEL
LIN {X 0,Y 474.606,Z 525.34,A -85,B 0,C 180,E1 -7422.234,E2 -7422.234} C_VEL
LIN {X 0,Y 474.621,Z 525.362,A -85,B 0,C 180,E1 -7425.298,E2 -7425.298} C_VEL
LIN {X 0,Y 474.625,Z 525.357,A -85,B 0,C 180,E1 -7428.214,E2 -7428.214} C_VEL
LIN {X 0,Y 474.615,Z 525.36,A -85,B 0,C 180,E1 -7431.542,E2 -7431.542} C_VEL
LIN {X 0,Y 474.61,Z 525.362,A -85,B 0,C 180,E1 -7435.025,E2 -7435.025} C_VEL
LIN {X 0,Y 473.933,Z 525.446,A -85,B 0,C 180,E1 -7435.733,E2 -7435.733} C_VEL
LIN {X 0,Y 471.079,Z 525.805,A -85,B 0,C 180,E1 -7436.884,E2 -7436.884} C_VEL
LIN {X 0,Y 468.675,Z 526.102,A -85,B 0,C 180,E1 -7437.812,E2 -7437.812} C_VEL
LIN {X 0,Y 467.65,Z 526.231,A -85,B 0,C 180,E1 -7438.529,E2 -7438.529} C_VEL
LIN {X 0,Y 467.57,Z 526.24,A -85,B 0,C 180,E1 -7438.771,E2 -7438.771} C_VEL
LIN {X 0,Y 467.625,Z 526.234,A -85,B 0,C 180,E1 -7442.231,E2 -7442.231} C_VEL
LIN {X 0,Y 467.597,Z 526.234,A -85,B 0,C 180,E1 -7445.112,E2 -7445.112} C_VEL
LIN {X 0,Y 467.625,Z 526.347,A -85,B 0,C 180,E1 -7448.026,E2 -7448.026} C_VEL
LIN {X 0,Y 469.06,Z 534.098,A -85,B 0,C 180,E1 -7449.841,E2 -7449.841} C_VEL
LIN {X 0,Y 468.491,Z 548.322,A -85,B 0,C 180,E1 -7452.877,E2 -7452.877} C_VEL
LIN {X 0,Y 468.55,Z 549.663,A -85,B 0,C 180,E1 -7453.048,E2 -7453.048} C_VEL
LIN {X 0,Y 471.402,Z 564.821,A -85,B 0,C 180,E1 -7453.404,E2 -7453.404} C_VEL
LIN {X 0,Y 470.665,Z 656.271,A -85,B 0,C 180,E1 -7454.824,E2 -7454.824} C_VEL
LIN {X 0,Y 470.337,Z 670.159,A -85,B 0,C 180,E1 -7455.228,E2 -7455.228} C_VEL
LIN {X 0,Y 469.954,Z 682.571,A -85,B 0,C 180,E1 -7455.769,E2 -7455.769} C_VEL
LIN {X 0,Y 469.47,Z 694.778,A -85,B 0,C 180,E1 -7456.497,E2 -7456.497} C_VEL
LIN {X 0,Y 469.032,Z 705.788,A -85,B 0,C 180,E1 -7457.341,E2 -7457.341} C_VEL
LIN {X 0,Y 468.498,Z 716.032,A -85,B 0,C 180,E1 -7458.315,E2 -7458.315} C_VEL
LIN {X 0,Y 468.062,Z 725.219,A -85,B 0,C 180,E1 -7459.4,E2 -7459.4} C_VEL
LIN {X 0,Y 467.624,Z 734.137,A -85,B 0,C 180,E1 -7460.702,E2 -7460.702} C_VEL
LIN {X 0,Y 467.236,Z 741.317,A -85,B 0,C 180,E1 -7462.002,E2 -7462.002} C_VEL
LIN {X 0,Y 467.021,Z 747.118,A -85,B 0,C 180,E1 -7463.319,E2 -7463.319} C_VEL
LIN {X 0,Y 466.923,Z 750.865,A -85,B 0,C 180,E1 -7464.385,E2 -7464.385} C_VEL
LIN {X 0,Y 466.771,Z 754.466,A -85,B 0,C 180,E1 -7465.682,E2 -7465.682} C_VEL
LIN {X 0,Y 466.774,Z 756.326,A -85,B 0,C 180,E1 -7466.546,E2 -7466.546} C_VEL
LIN {X 0,Y 466.684,Z 757.732,A -85,B 0,C 180,E1 -7467.41,E2 -7467.41} C_VEL
LIN {X 0,Y 466.62,Z 759.348,A -85,B 0,C 180,E1 -7469.136,E2 -7469.136} C_VEL
LIN {X 0,Y 466.599,Z 759.585,A -85,B 0,C 180,E1 -7469.999,E2 -7469.999} C_VEL
LIN {X 0,Y 466.619,Z 759.399,A -85,B 0,C 180,E1 -7470.862,E2 -7470.862} C_VEL
LIN {X 0,Y 466.684,Z 757.853,A -85,B 0,C 180,E1 -7472.589,E2 -7472.589} C_VEL
LIN {X 0,Y 466.774,Z 756.498,A -85,B 0,C 180,E1 -7473.452,E2 -7473.452} C_VEL
LIN {X 0,Y 466.744,Z 753.636,A -85,B 0,C 180,E1 -7474.75,E2 -7474.75} C_VEL
LIN {X 0,Y 466.992,Z 749.748,A -85,B 0,C 180,E1 -7476.046,E2 -7476.046} C_VEL
LIN {X 0,Y 467.096,Z 744.743,A -85,B 0,C 180,E1 -7477.347,E2 -7477.347} C_VEL
LIN {X 0,Y 467.407,Z 738.438,A -85,B 0,C 180,E1 -7478.647,E2 -7478.647} C_VEL
LIN {X 0,Y 467.752,Z 730.543,A -85,B 0,C 180,E1 -7479.949,E2 -7479.949} C_VEL
LIN {X 0,Y 468.131,Z 722.495,A -85,B 0,C 180,E1 -7481.034,E2 -7481.034} C_VEL
LIN {X 0,Y 468.722,Z 712.666,A -85,B 0,C 180,E1 -7482.117,E2 -7482.117} C_VEL
LIN {X 0,Y 469.187,Z 701.484,A -85,B 0,C 180,E1 -7483.105,E2 -7483.105} C_VEL
LIN {X 0,Y 469.622,Z 690.795,A -85,B 0,C 180,E1 -7483.853,E2 -7483.853} C_VEL
LIN {X 0,Y 470.122,Z 678.824,A -85,B 0,C 180,E1 -7484.5,E2 -7484.5} C_VEL
LIN {X 0,Y 470.468,Z 665.713,A -85,B 0,C 180,E1 -7485.015,E2 -7485.015} C_VEL
LIN {X 0,Y 470.741,Z 652.544,A -85,B 0,C 180,E1 -7485.338,E2 -7485.338} C_VEL
LIN {X 0,Y 471.241,Z 563.681,A -85,B 0,C 180,E1 -7486.711,E2 -7486.711} C_VEL
LIN {X 0,Y 468.497,Z 549.402,A -85,B 0,C 180,E1 -7487.061,E2 -7487.061} C_VEL
LIN {X 0,Y 468.541,Z 547.152,A -85,B 0,C 180,E1 -7487.456,E2 -7487.456} C_VEL
LIN {X 0,Y 469.067,Z 534.504,A -85,B 0,C 180,E1 -7490.157,E2 -7490.157} C_VEL
LIN {X 0,Y 467.604,Z 526.291,A -85,B 0,C 180,E1 -7492.098,E2 -7492.098} C_VEL
LIN {X 0,Y 467.614,Z 526.233,A -85,B 0,C 180,E1 -7495.608,E2 -7495.608} C_VEL
LIN {X 0,Y 467.627,Z 526.235,A -85,B 0,C 180,E1 -7497.768,E2 -7497.768} C_VEL
LIN {X 0,Y 467.568,Z 526.24,A -85,B 0,C 180,E1 -7501.044,E2 -7501.044} C_VEL
LIN {X 0,Y 467.588,Z 526.238,A -85,B 0,C 180,E1 -7504.242,E2 -7504.242} C_VEL
LIN {X 0,Y 467.548,Z 526.244,A -85,B 0,C 180,E1 -7507.186,E2 -7507.186} C_VEL
LIN {X 0,Y 467.576,Z 526.234,A -85,B 0,C 180,E1 -7510.263,E2 -7510.263} C_VEL
LIN {X 0,Y 467.583,Z 526.238,A -85,B 0,C 180,E1 -7512.566,E2 -7512.566} C_VEL
LIN {X 0,Y 467.566,Z 526.235,A -85,B 0,C 180,E1 -7515.052,E2 -7515.052} C_VEL
LIN {X 0,Y 467.584,Z 526.243,A -85,B 0,C 180,E1 -7517.439,E2 -7517.439} C_VEL
LIN {X 0,Y 467.614,Z 526.227,A -85,B 0,C 180,E1 -7520.858,E2 -7520.858} C_VEL
LIN {X 0,Y 467.558,Z 526.24,A -85,B 0,C 180,E1 -7524.259,E2 -7524.259} C_VEL
LIN {X 0,Y 467.577,Z 526.242,A -85,B 0,C 180,E1 -7527.32,E2 -7527.32} C_VEL
LIN {X 0,Y 467.572,Z 526.238,A -85,B 0,C 180,E1 -7530.665,E2 -7530.665} C_VEL
LIN {X 0,Y 467.621,Z 526.231,A -85,B 0,C 180,E1 -7533.2,E2 -7533.2} C_VEL
LIN {X 0,Y 467.586,Z 526.234,A -85,B 0,C 180,E1 -7536.468,E2 -7536.468} C_VEL
LIN {X 0,Y 467.617,Z 526.237,A -85,B 0,C 180,E1 -7539.777,E2 -7539.777} C_VEL
LIN {X 0,Y 467.602,Z 526.231,A -85,B 0,C 180,E1 -7542.506,E2 -7542.506} C_VEL
LIN {X 0,Y 467.599,Z 526.234,A -85,B 0,C 180,E1 -7545.196,E2 -7545.196} C_VEL
LIN {X 0,Y 467.648,Z 526.23,A -85,B 0,C 180,E1 -7547.854,E2 -7547.854} C_VEL
LIN {X 0,Y 467.675,Z 526.225,A -85,B 0,C 180,E1 -7551.357,E2 -7551.357} C_VEL
LIN {X 0,Y 467.737,Z 526.22,A -85,B 0,C 180,E1 -7553.962,E2 -7553.962} C_VEL
LIN {X 0,Y 467.853,Z 526.202,A -85,B 0,C 180,E1 -7557.417,E2 -7557.417} C_VEL
LIN {X 0,Y 467.875,Z 526.203,A -85,B 0,C 180,E1 -7560,E2 -7560} C_VEL
LIN {X 0,Y 467.853,Z 526.199,A -85,B 0,C 180,E1 -7562.583,E2 -7562.583} C_VEL
LIN {X 0,Y 467.736,Z 526.22,A -85,B 0,C 180,E1 -7566.037,E2 -7566.037} C_VEL
LIN {X 0,Y 467.674,Z 526.223,A -85,B 0,C 180,E1 -7568.643,E2 -7568.643} C_VEL
LIN {X 0,Y 467.675,Z 526.226,A -85,B 0,C 180,E1 -7572.145,E2 -7572.145} C_VEL
LIN {X 0,Y 467.642,Z 526.229,A -85,B 0,C 180,E1 -7575.886,E2 -7575.886} C_VEL
LIN {X 0,Y 467.617,Z 526.237,A -85,B 0,C 180,E1 -7579.308,E2 -7579.308} C_VEL
LIN {X 0,Y 467.53,Z 526.244,A -85,B 0,C 180,E1 -7582.074,E2 -7582.074} C_VEL
LIN {X 0,Y 467.597,Z 526.236,A -85,B 0,C 180,E1 -7584.888,E2 -7584.888} C_VEL
LIN {X 0,Y 467.621,Z 526.239,A -85,B 0,C 180,E1 -7587.769,E2 -7587.769} C_VEL
LIN {X 0,Y 467.563,Z 526.238,A -85,B 0,C 180,E1 -7591.046,E2 -7591.046} C_VEL
LIN {X 0,Y 467.584,Z 526.236,A -85,B 0,C 180,E1 -7594.243,E2 -7594.243} C_VEL
LIN {X 0,Y 467.545,Z 526.233,A -85,B 0,C 180,E1 -7597.188,E2 -7597.188} C_VEL
LIN {X 0,Y 467.572,Z 526.239,A -85,B 0,C 180,E1 -7600.265,E2 -7600.265} C_VEL
LIN {X 0,Y 467.581,Z 526.23,A -85,B 0,C 180,E1 -7602.568,E2 -7602.568} C_VEL
LIN {X 0,Y 467.566,Z 526.241,A -85,B 0,C 180,E1 -7605.054,E2 -7605.054} C_VEL
LIN {X 0,Y 467.62,Z 526.232,A -85,B 0,C 180,E1 -7607.445,E2 -7607.445} C_VEL
LIN {X 0,Y 467.612,Z 526.23,A -85,B 0,C 180,E1 -7610.86,E2 -7610.86} C_VEL
LIN {X 0,Y 467.56,Z 526.243,A -85,B 0,C 180,E1 -7614.261,E2 -7614.261} C_VEL
LIN {X 0,Y 467.58,Z 526.219,A -85,B 0,C 180,E1 -7617.322,E2 -7617.322} C_VEL
LIN {X 0,Y 467.569,Z 526.232,A -85,B 0,C 180,E1 -7620.668,E2 -7620.668} C_VEL
LIN {X 0,Y 467.616,Z 526.218,A -85,B 0,C 180,E1 -7623.201,E2 -7623.201} C_VEL
LIN {X 0,Y 467.676,Z 526.43,A -85,B 0,C 180,E1 -7624.242,E2 -7624.242} C_VEL
LIN {X 0,Y 469.754,Z 537.36,A -85,B 0,C 180,E1 -7626.41,E2 -7626.41} C_VEL
LIN {X 0,Y 469.657,Z 544.976,A -85,B 0,C 180,E1 -7627.801,E2 -7627.801} C_VEL
LIN {X 0,Y 468.882,Z 561.651,A -85,B 0,C 180,E1 -7630.787,E2 -7630.787} C_VEL
LIN {X 0,Y 468.441,Z 574.148,A -85,B 0,C 180,E1 -7632.965,E2 -7632.965} C_VEL
LIN {X 0,Y 471.248,Z 591.953,A -85,B 0,C 180,E1 -7633.37,E2 -7633.37} C_VEL
LIN {X 0,Y 470.598,Z 682.117,A -85,B 0,C 180,E1 -7634.768,E2 -7634.768} C_VEL
LIN {X 0,Y 470.24,Z 695.377,A -85,B 0,C 180,E1 -7635.144,E2 -7635.144} C_VEL
LIN {X 0,Y 469.825,Z 707.542,A -85,B 0,C 180,E1 -7635.656,E2 -7635.656} C_VEL
LIN {X 0,Y 469.33,Z 719.828,A -85,B 0,C 180,E1 -7636.359,E2 -7636.359} C_VEL
LIN {X 0,Y 468.774,Z 731.007,A -85,B 0,C 180,E1 -7637.19,E2 -7637.19} C_VEL
LIN {X 0,Y 468.306,Z 741.868,A -85,B 0,C 180,E1 -7638.202,E2 -7638.202} C_VEL
LIN {X 0,Y 467.823,Z 750.408,A -85,B 0,C 180,E1 -7639.177,E2 -7639.177} C_VEL
LIN {X 0,Y 467.477,Z 758.29,A -85,B 0,C 180,E1 -7640.264,E2 -7640.264} C_VEL
LIN {X 0,Y 467.13,Z 765.989,A -85,B 0,C 180,E1 -7641.566,E2 -7641.566} C_VEL
LIN {X 0,Y 466.858,Z 773.085,A -85,B 0,C 180,E1 -7643.084,E2 -7643.084} C_VEL
LIN {X 0,Y 466.783,Z 777.809,A -85,B 0,C 180,E1 -7644.385,E2 -7644.385} C_VEL
LIN {X 0,Y 466.652,Z 781.42,A -85,B 0,C 180,E1 -7645.682,E2 -7645.682} C_VEL
LIN {X 0,Y 466.691,Z 783.284,A -85,B 0,C 180,E1 -7646.547,E2 -7646.547} C_VEL
LIN {X 0,Y 466.661,Z 784.679,A -85,B 0,C 180,E1 -7647.411,E2 -7647.411} C_VEL
LIN {X 0,Y 466.618,Z 786.28,A -85,B 0,C 180,E1 -7649.138,E2 -7649.138} C_VEL
LIN {X 0,Y 466.598,Z 786.495,A -85,B 0,C 180,E1 -7650.001,E2 -7650.001} C_VEL
LIN {X 0,Y 466.618,Z 786.278,A -85,B 0,C 180,E1 -7650.864,E2 -7650.864} C_VEL
LIN {X 0,Y 466.662,Z 784.674,A -85,B 0,C 180,E1 -7652.59,E2 -7652.59} C_VEL
LIN {X 0,Y 466.691,Z 783.278,A -85,B 0,C 180,E1 -7653.454,E2 -7653.454} C_VEL
LIN {X 0,Y 466.695,Z 780.343,A -85,B 0,C 180,E1 -7654.752,E2 -7654.752} C_VEL
LIN {X 0,Y 466.782,Z 776.372,A -85,B 0,C 180,E1 -7656.051,E2 -7656.051} C_VEL
LIN {X 0,Y 466.98,Z 770.259,A -85,B 0,C 180,E1 -7657.568,E2 -7657.568} C_VEL
LIN {X 0,Y 467.242,Z 763.581,A -85,B 0,C 180,E1 -7658.87,E2 -7658.87} C_VEL
LIN {X 0,Y 467.597,Z 755.296,A -85,B 0,C 180,E1 -7660.173,E2 -7660.173} C_VEL
LIN {X 0,Y 468.025,Z 746.806,A -85,B 0,C 180,E1 -7661.258,E2 -7661.258} C_VEL
LIN {X 0,Y 468.589,Z 736.646,A -85,B 0,C 180,E1 -7662.311,E2 -7662.311} C_VEL
LIN {X 0,Y 468.949,Z 725.933,A -85,B 0,C 180,E1 -7663.212,E2 -7663.212} C_VEL
LIN {X 0,Y 469.501,Z 714.564,A -85,B 0,C 180,E1 -7663.968,E2 -7663.968} C_VEL
LIN {X 0,Y 469.988,Z 702.903,A -85,B 0,C 180,E1 -7664.561,E2 -7664.561} C_VEL
LIN {X 0,Y 470.415,Z 689.452,A -85,B 0,C 180,E1 -7665.046,E2 -7665.046} C_VEL
LIN {X 0,Y 470.693,Z 676.149,A -85,B 0,C 180,E1 -7665.342,E2 -7665.342} C_VEL
LIN {X 0,Y 471.101,Z 590.845,A -85,B 0,C 180,E1 -7666.652,E2 -7666.652} C_VEL
LIN {X 0,Y 468.447,Z 574.284,A -85,B 0,C 180,E1 -7667.025,E2 -7667.025} C_VEL
LIN {X 0,Y 468.587,Z 568.965,A -85,B 0,C 180,E1 -7667.907,E2 -7667.907} C_VEL
LIN {X 0,Y 469.316,Z 552.563,A -85,B 0,C 180,E1 -7670.834,E2 -7670.834} C_VEL
LIN {X 0,Y 469.904,Z 538.612,A -85,B 0,C 180,E1 -7673.35,E2 -7673.35} C_VEL
LIN {X 0,Y 467.753,Z 526.855,A -85,B 0,C 180,E1 -7675.644,E2 -7675.644} C_VEL
LIN {X 0,Y 467.652,Z 526.254,A -85,B 0,C 180,E1 -7675.838,E2 -7675.838} C_VEL
LIN {X 0,Y 467.58,Z 526.226,A -85,B 0,C 180,E1 -7678.75,E2 -7678.75} C_VEL
LIN {X 0,Y 467.587,Z 526.241,A -85,B 0,C 180,E1 -7681.74,E2 -7681.74} C_VEL
LIN {X 0,Y 467.568,Z 526.24,A -85,B 0,C 180,E1 -7684.833,E2 -7684.833} C_VEL
LIN {X 0,Y 467.569,Z 526.245,A -85,B 0,C 180,E1 -7688.045,E2 -7688.045} C_VEL
LIN {X 0,Y 467.582,Z 526.239,A -85,B 0,C 180,E1 -7691.277,E2 -7691.277} C_VEL
LIN {X 0,Y 467.556,Z 526.245,A -85,B 0,C 180,E1 -7693.821,E2 -7693.821} C_VEL
LIN {X 0,Y 467.557,Z 526.245,A -85,B 0,C 180,E1 -7696.256,E2 -7696.256} C_VEL
LIN {X 0,Y 467.581,Z 526.24,A -85,B 0,C 180,E1 -7698.723,E2 -7698.723} C_VEL
LIN {X 0,Y 467.569,Z 526.245,A -85,B 0,C 180,E1 -7701.956,E2 -7701.956} C_VEL
LIN {X 0,Y 467.571,Z 526.241,A -85,B 0,C 180,E1 -7705.168,E2 -7705.168} C_VEL
LIN {X 0,Y 467.586,Z 526.243,A -85,B 0,C 180,E1 -7708.26,E2 -7708.26} C_VEL
LIN {X 0,Y 467.58,Z 526.242,A -85,B 0,C 180,E1 -7711.251,E2 -7711.251} C_VEL
LIN {X 0,Y 467.725,Z 526.431,A -85,B 0,C 180,E1 -7713.15,E2 -7713.15} C_VEL
LIN {X 0,Y 469.937,Z 538.115,A -85,B 0,C 180,E1 -7715.008,E2 -7715.008} C_VEL
LIN {X 0,Y 469.593,Z 555.525,A -85,B 0,C 180,E1 -7717.565,E2 -7717.565} C_VEL
LIN {X 0,Y 469.041,Z 575.583,A -85,B 0,C 180,E1 -7720.548,E2 -7720.548} C_VEL
LIN {X 0,Y 468.49,Z 598.2,A -85,B 0,C 180,E1 -7723.908,E2 -7723.908} C_VEL
LIN {X 0,Y 468.048,Z 616.796,A -85,B 0,C 180,E1 -7726.655,E2 -7726.655} C_VEL
LIN {X 0,Y 469.465,Z 628.993,A -85,B 0,C 180,E1 -7726.933,E2 -7726.933} C_VEL
LIN {X 0,Y 468.959,Z 696.577,A -85,B 0,C 180,E1 -7728.108,E2 -7728.108} C_VEL
LIN {X 0,Y 468.724,Z 706.494,A -85,B 0,C 180,E1 -7728.404,E2 -7728.404} C_VEL
LIN {X 0,Y 468.532,Z 715.941,A -85,B 0,C 180,E1 -7728.81,E2 -7728.81} C_VEL
LIN {X 0,Y 468.279,Z 726.309,A -85,B 0,C 180,E1 -7729.406,E2 -7729.406} C_VEL
LIN {X 0,Y 467.927,Z 736.232,A -85,B 0,C 180,E1 -7730.163,E2 -7730.163} C_VEL
LIN {X 0,Y 467.645,Z 744.088,A -85,B 0,C 180,E1 -7730.921,E2 -7730.921} C_VEL
LIN {X 0,Y 467.323,Z 751.437,A -85,B 0,C 180,E1 -7731.786,E2 -7731.786} C_VEL
LIN {X 0,Y 467.143,Z 757.493,A -85,B 0,C 180,E1 -7732.653,E2 -7732.653} C_VEL
LIN {X 0,Y 467.042,Z 762.836,A -85,B 0,C 180,E1 -7733.579,E2 -7733.579} C_VEL
LIN {X 0,Y 466.826,Z 768.578,A -85,B 0,C 180,E1 -7734.817,E2 -7734.817} C_VEL
LIN {X 0,Y 466.78,Z 772.924,A -85,B 0,C 180,E1 -7736.115,E2 -7736.115} C_VEL
LIN {X 0,Y 466.669,Z 775.93,A -85,B 0,C 180,E1 -7737.411,E2 -7737.411} C_VEL
LIN {X 0,Y 466.607,Z 777.271,A -85,B 0,C 180,E1 -7738.274,E2 -7738.274} C_VEL
LIN {X 0,Y 466.588,Z 778.108,A -85,B 0,C 180,E1 -7739.137,E2 -7739.137} C_VEL
LIN {X 0,Y 466.597,Z 778.412,A -85,B 0,C 180,E1 -7740,E2 -7740} C_VEL
LIN {X 0,Y 466.589,Z 778.133,A -85,B 0,C 180,E1 -7740.863,E2 -7740.863} C_VEL
LIN {X 0,Y 466.608,Z 777.352,A -85,B 0,C 180,E1 -7741.726,E2 -7741.726} C_VEL
LIN {X 0,Y 466.669,Z 776.072,A -85,B 0,C 180,E1 -7742.59,E2 -7742.59} C_VEL
LIN {X 0,Y 466.778,Z 773.126,A -85,B 0,C 180,E1 -7743.885,E2 -7743.885} C_VEL
LIN {X 0,Y 466.818,Z 768.885,A -85,B 0,C 180,E1 -7745.183,E2 -7745.183} C_VEL
LIN {X 0,Y 466.99,Z 763.456,A -85,B 0,C 180,E1 -7746.387,E2 -7746.387} C_VEL
LIN {X 0,Y 467.129,Z 758.034,A -85,B 0,C 180,E1 -7747.347,E2 -7747.347} C_VEL
LIN {X 0,Y 467.316,Z 752.093,A -85,B 0,C 180,E1 -7748.214,E2 -7748.214} C_VEL
LIN {X 0,Y 467.605,Z 744.889,A -85,B 0,C 180,E1 -7749.08,E2 -7749.08} C_VEL
LIN {X 0,Y 467.976,Z 736.04,A -85,B 0,C 180,E1 -7749.945,E2 -7749.945} C_VEL
LIN {X 0,Y 468.287,Z 726.072,A -85,B 0,C 180,E1 -7750.703,E2 -7750.703} C_VEL
LIN {X 0,Y 468.576,Z 715.684,A -85,B 0,C 180,E1 -7751.299,E2 -7751.299} C_VEL
LIN {X 0,Y 468.736,Z 706.186,A -85,B 0,C 180,E1 -7751.706,E2 -7751.706} C_VEL
LIN {X 0,Y 468.965,Z 695.132,A -85,B 0,C 180,E1 -7752.029,E2 -7752.029} C_VEL
LIN {X 0,Y 469.379,Z 627.896,A -85,B 0,C 180,E1 -7753.159,E2 -7753.159} C_VEL
LIN {X 0,Y 468.022,Z 616.604,A -85,B 0,C 180,E1 -7753.407,E2 -7753.407} C_VEL
LIN {X 0,Y 468.506,Z 597.354,A -85,B 0,C 180,E1 -7756.326,E2 -7756.326} C_VEL
LIN {X 0,Y 469.184,Z 575.332,A -85,B 0,C 180,E1 -7759.696,E2 -7759.696} C_VEL
LIN {X 0,Y 469.816,Z 556.07,A -85,B 0,C 180,E1 -7762.656,E2 -7762.656} C_VEL
LIN {X 0,Y 470.331,Z 541.046,A -85,B 0,C 180,E1 -7764.969,E2 -7764.969} C_VEL
LIN {X 0,Y 469.314,Z 534.477,A -85,B 0,C 180,E1 -7766.037,E2 -7766.037} C_VEL
LIN {X 0,Y 467.665,Z 526.329,A -85,B 0,C 180,E1 -7767.428,E2 -7767.428} C_VEL
LIN {X 0,Y 467.572,Z 526.242,A -85,B 0,C 180,E1 -7771.045,E2 -7771.045} C_VEL
LIN {X 0,Y 467.593,Z 526.238,A -85,B 0,C 180,E1 -7774.242,E2 -7774.242} C_VEL
LIN {X 0,Y 467.552,Z 526.245,A -85,B 0,C 180,E1 -7777.186,E2 -7777.186} C_VEL
LIN {X 0,Y 467.581,Z 526.227,A -85,B 0,C 180,E1 -7780.264,E2 -7780.264} C_VEL
LIN {X 0,Y 467.552,Z 526.233,A -85,B 0,C 180,E1 -7783.745,E2 -7783.745} C_VEL
LIN {X 0,Y 467.558,Z 526.241,A -85,B 0,C 180,E1 -7786.255,E2 -7786.255} C_VEL
LIN {X 0,Y 467.582,Z 526.236,A -85,B 0,C 180,E1 -7788.723,E2 -7788.723} C_VEL
LIN {X 0,Y 467.568,Z 526.237,A -85,B 0,C 180,E1 -7791.955,E2 -7791.955} C_VEL
LIN {X 0,Y 467.562,Z 526.241,A -85,B 0,C 180,E1 -7795.167,E2 -7795.167} C_VEL
LIN {X 0,Y 467.587,Z 526.237,A -85,B 0,C 180,E1 -7798.26,E2 -7798.26} C_VEL
LIN {X 0,Y 467.57,Z 526.24,A -85,B 0,C 180,E1 -7798.771,E2 -7798.771} C_VEL
LIN {X 0,Y 466.916,Z 526.326,A -85,B 0,C 180,E1 -7799.49,E2 -7799.49} C_VEL
LIN {X 0,Y 464.085,Z 526.679,A -85,B 0,C 180,E1 -7800.657,E2 -7800.657} C_VEL
LIN {X 0,Y 461.687,Z 526.974,A -85,B 0,C 180,E1 -7801.598,E2 -7801.598} C_VEL
LIN {X 0,Y 460.659,Z 527.103,A -85,B 0,C 180,E1 -7802.325,E2 -7802.325} C_VEL
LIN {X 0,Y 460.576,Z 527.115,A -85,B 0,C 180,E1 -7802.571,E2 -7802.571} C_VEL
LIN {X 0,Y 460.541,Z 527.109,A -85,B 0,C 180,E1 -7805.667,E2 -7805.667} C_VEL
LIN {X 0,Y 460.572,Z 527.326,A -85,B 0,C 180,E1 -7807.869,E2 -7807.869} C_VEL
LIN {X 0,Y 462.1,Z 535.309,A -85,B 0,C 180,E1 -7809.756,E2 -7809.756} C_VEL
LIN {X 0,Y 461.556,Z 549.274,A -85,B 0,C 180,E1 -7812.737,E2 -7812.737} C_VEL
LIN {X 0,Y 462.184,Z 552.75,A -85,B 0,C 180,E1 -7812.866,E2 -7812.866} C_VEL
LIN {X 0,Y 464.608,Z 566.167,A -85,B 0,C 180,E1 -7813.172,E2 -7813.172} C_VEL
LIN {X 0,Y 463.837,Z 656.495,A -85,B 0,C 180,E1 -7814.595,E2 -7814.595} C_VEL
LIN {X 0,Y 463.494,Z 670.376,A -85,B 0,C 180,E1 -7815.005,E2 -7815.005} C_VEL
LIN {X 0,Y 463.08,Z 682.784,A -85,B 0,C 180,E1 -7815.553,E2 -7815.553} C_VEL
LIN {X 0,Y 462.597,Z 694.636,A -85,B 0,C 180,E1 -7816.268,E2 -7816.268} C_VEL
LIN {X 0,Y 462.111,Z 705.998,A -85,B 0,C 180,E1 -7817.148,E2 -7817.148} C_VEL
LIN {X 0,Y 461.556,Z 716.242,A -85,B 0,C 180,E1 -7818.137,E2 -7818.137} C_VEL
LIN {X 0,Y 461.082,Z 725.427,A -85,B 0,C 180,E1 -7819.238,E2 -7819.238} C_VEL
LIN {X 0,Y 460.598,Z 734.346,A -85,B 0,C 180,E1 -7820.559,E2 -7820.559} C_VEL
LIN {X 0,Y 460.212,Z 741.524,A -85,B 0,C 180,E1 -7821.879,E2 -7821.879} C_VEL
LIN {X 0,Y 459.939,Z 747.726,A -85,B 0,C 180,E1 -7823.325,E2 -7823.325} C_VEL
LIN {X 0,Y 459.744,Z 752.388,A -85,B 0,C 180,E1 -7824.737,E2 -7824.737} C_VEL
LIN {X 0,Y 459.676,Z 754.672,A -85,B 0,C 180,E1 -7825.615,E2 -7825.615} C_VEL
LIN {X 0,Y 459.707,Z 756.531,A -85,B 0,C 180,E1 -7826.493,E2 -7826.493} C_VEL
LIN {X 0,Y 459.608,Z 757.937,A -85,B 0,C 180,E1 -7827.37,E2 -7827.37} C_VEL
LIN {X 0,Y 459.523,Z 759.553,A -85,B 0,C 180,E1 -7829.123,E2 -7829.123} C_VEL
LIN {X 0,Y 459.53,Z 759.789,A -85,B 0,C 180,E1 -7829.999,E2 -7829.999} C_VEL
LIN {X 0,Y 459.523,Z 759.604,A -85,B 0,C 180,E1 -7830.876,E2 -7830.876} C_VEL
LIN {X 0,Y 459.608,Z 758.057,A -85,B 0,C 180,E1 -7832.629,E2 -7832.629} C_VEL
LIN {X 0,Y 459.688,Z 756.702,A -85,B 0,C 180,E1 -7833.505,E2 -7833.505} C_VEL
LIN {X 0,Y 459.67,Z 753.84,A -85,B 0,C 180,E1 -7834.823,E2 -7834.823} C_VEL
LIN {X 0,Y 459.92,Z 749.951,A -85,B 0,C 180,E1 -7836.14,E2 -7836.14} C_VEL
LIN {X 0,Y 460.045,Z 744.946,A -85,B 0,C 180,E1 -7837.46,E2 -7837.46} C_VEL
LIN {X 0,Y 460.377,Z 738.64,A -85,B 0,C 180,E1 -7838.78,E2 -7838.78} C_VEL
LIN {X 0,Y 460.759,Z 730.744,A -85,B 0,C 180,E1 -7840.102,E2 -7840.102} C_VEL
LIN {X 0,Y 461.259,Z 720.921,A -85,B 0,C 180,E1 -7841.424,E2 -7841.424} C_VEL
LIN {X 0,Y 461.919,Z 710.626,A -85,B 0,C 180,E1 -7842.519,E2 -7842.519} C_VEL
LIN {X 0,Y 462.354,Z 699.538,A -85,B 0,C 180,E1 -7843.471,E2 -7843.471} C_VEL
LIN {X 0,Y 462.845,Z 689.228,A -85,B 0,C 180,E1 -7844.172,E2 -7844.172} C_VEL
LIN {X 0,Y 463.276,Z 677.891,A -85,B 0,C 180,E1 -7844.776,E2 -7844.776} C_VEL
LIN {X 0,Y 463.671,Z 664.988,A -85,B 0,C 180,E1 -7845.269,E2 -7845.269} C_VEL
LIN {X 0,Y 463.946,Z 651.22,A -85,B 0,C 180,E1 -7845.597,E2 -7845.597} C_VEL
LIN {X 0,Y 464.441,Z 564.49,A -85,B 0,C 180,E1 -7846.953,E2 -7846.953} C_VEL
LIN {X 0,Y 461.566,Z 549.626,A -85,B 0,C 180,E1 -7847.324,E2 -7847.324} C_VEL
LIN {X 0,Y 461.59,Z 547.342,A -85,B 0,C 180,E1 -7847.728,E2 -7847.728} C_VEL
LIN {X 0,Y 462.107,Z 535.732,A -85,B 0,C 180,E1 -7850.242,E2 -7850.242} C_VEL
LIN {X 0,Y 460.561,Z 527.143,A -85,B 0,C 180,E1 -7852.308,E2 -7852.308} C_VEL
LIN {X 0,Y 460.567,Z 527.109,A -85,B 0,C 180,E1 -7855.801,E2 -7855.801} C_VEL
LIN {X 0,Y 460.555,Z 527.113,A -85,B 0,C 180,E1 -7858.232,E2 -7858.232} C_VEL
LIN {X 0,Y 460.521,Z 527.121,A -85,B 0,C 180,E1 -7861.282,E2 -7861.282} C_VEL
LIN {X 0,Y 460.532,Z 527.117,A -85,B 0,C 180,E1 -7864.505,E2 -7864.505} C_VEL
LIN {X 0,Y 460.526,Z 527.122,A -85,B 0,C 180,E1 -7867.619,E2 -7867.619} C_VEL
LIN {X 0,Y 460.54,Z 527.111,A -85,B 0,C 180,E1 -7870.269,E2 -7870.269} C_VEL
LIN {X 0,Y 460.506,Z 527.122,A -85,B 0,C 180,E1 -7873.373,E2 -7873.373} C_VEL
LIN {X 0,Y 460.495,Z 527.118,A -85,B 0,C 180,E1 -7876.624,E2 -7876.624} C_VEL
LIN {X 0,Y 460.554,Z 527.11,A -85,B 0,C 180,E1 -7879.727,E2 -7879.727} C_VEL
LIN {X 0,Y 460.524,Z 527.109,A -85,B 0,C 180,E1 -7882.518,E2 -7882.518} C_VEL
LIN {X 0,Y 460.543,Z 527.119,A -85,B 0,C 180,E1 -7885.623,E2 -7885.623} C_VEL
LIN {X 0,Y 460.531,Z 527.114,A -85,B 0,C 180,E1 -7888.744,E2 -7888.744} C_VEL
LIN {X 0,Y 460.553,Z 527.112,A -85,B 0,C 180,E1 -7891.767,E2 -7891.767} C_VEL
LIN {X 0,Y 460.553,Z 527.113,A -85,B 0,C 180,E1 -7894.705,E2 -7894.705} C_VEL
LIN {X 0,Y 460.505,Z 527.119,A -85,B 0,C 180,E1 -7897.571,E2 -7897.571} C_VEL
LIN {X 0,Y 460.563,Z 527.111,A -85,B 0,C 180,E1 -7900.384,E2 -7900.384} C_VEL
LIN {X 0,Y 460.558,Z 527.112,A -85,B 0,C 180,E1 -7903.146,E2 -7903.146} C_VEL
LIN {X 0,Y 460.548,Z 527.116,A -85,B 0,C 180,E1 -7905.868,E2 -7905.868} C_VEL
LIN {X 0,Y 460.604,Z 527.104,A -85,B 0,C 180,E1 -7908.559,E2 -7908.559} C_VEL
LIN {X 0,Y 460.687,Z 527.096,A -85,B 0,C 180,E1 -7912.108,E2 -7912.108} C_VEL
LIN {X 0,Y 460.691,Z 527.095,A -85,B 0,C 180,E1 -7914.748,E2 -7914.748} C_VEL
LIN {X 0,Y 460.818,Z 527.078,A -85,B 0,C 180,E1 -7917.378,E2 -7917.378} C_VEL
LIN {X 0,Y 460.846,Z 527.078,A -85,B 0,C 180,E1 -7920,E2 -7920} C_VEL
LIN {X 0,Y 460.818,Z 527.076,A -85,B 0,C 180,E1 -7922.622,E2 -7922.622} C_VEL
LIN {X 0,Y 460.702,Z 527.095,A -85,B 0,C 180,E1 -7926.13,E2 -7926.13} C_VEL
LIN {X 0,Y 460.621,Z 527.102,A -85,B 0,C 180,E1 -7928.776,E2 -7928.776} C_VEL
LIN {X 0,Y 460.626,Z 527.103,A -85,B 0,C 180,E1 -7932.457,E2 -7932.457} C_VEL
LIN {X 0,Y 460.592,Z 527.106,A -85,B 0,C 180,E1 -7935.998,E2 -7935.998} C_VEL
LIN {X 0,Y 460.564,Z 527.112,A -85,B 0,C 180,E1 -7938.902,E2 -7938.902} C_VEL
LIN {X 0,Y 460.509,Z 527.12,A -85,B 0,C 180,E1 -7941.486,E2 -7941.486} C_VEL
LIN {X 0,Y 460.536,Z 527.115,A -85,B 0,C 180,E1 -7944.333,E2 -7944.333} C_VEL
LIN {X 0,Y 460.577,Z 527.108,A -85,B 0,C 180,E1 -7947.244,E2 -7947.244} C_VEL
LIN {X 0,Y 460.504,Z 527.118,A -85,B 0,C 180,E1 -7950.241,E2 -7950.241} C_VEL
LIN {X 0,Y 460.523,Z 527.12,A -85,B 0,C 180,E1 -7953.325,E2 -7953.325} C_VEL
LIN {X 0,Y 460.473,Z 527.111,A -85,B 0,C 180,E1 -7956.53,E2 -7956.53} C_VEL
LIN {X 0,Y 460.553,Z 527.118,A -85,B 0,C 180,E1 -7959.86,E2 -7959.86} C_VEL
LIN {X 0,Y 460.508,Z 527.112,A -85,B 0,C 180,E1 -7962.901,E2 -7962.901} C_VEL
LIN {X 0,Y 460.52,Z 527.119,A -85,B 0,C 180,E1 -7965.83,E2 -7965.83} C_VEL
LIN {X 0,Y 460.539,Z 527.116,A -85,B 0,C 180,E1 -7968.991,E2 -7968.991} C_VEL
LIN {X 0,Y 460.541,Z 527.11,A -85,B 0,C 180,E1 -7971.27,E2 -7971.27} C_VEL
LIN {X 0,Y 460.51,Z 527.12,A -85,B 0,C 180,E1 -7974.556,E2 -7974.556} C_VEL
LIN {X 0,Y 460.53,Z 527.086,A -85,B 0,C 180,E1 -7977.717,E2 -7977.717} C_VEL
LIN {X 0,Y 460.538,Z 527.109,A -85,B 0,C 180,E1 -7980.77,E2 -7980.77} C_VEL
LIN {X 0,Y 460.604,Z 527.13,A -85,B 0,C 180,E1 -7983.94,E2 -7983.94} C_VEL
LIN {X 0,Y 460.732,Z 527.841,A -85,B 0,C 180,E1 -7984.156,E2 -7984.156} C_VEL
LIN {X 0,Y 462.953,Z 539.726,A -85,B 0,C 180,E1 -7986.517,E2 -7986.517} C_VEL
LIN {X 0,Y 462.38,Z 553.662,A -85,B 0,C 180,E1 -7989.073,E2 -7989.073} C_VEL
LIN {X 0,Y 461.456,Z 573.253,A -85,B 0,C 180,E1 -7992.61,E2 -7992.61} C_VEL
LIN {X 0,Y 461.505,Z 574.332,A -85,B 0,C 180,E1 -7992.719,E2 -7992.719} C_VEL
LIN {X 0,Y 464.473,Z 592.981,A -85,B 0,C 180,E1 -7993.139,E2 -7993.139} C_VEL
LIN {X 0,Y 463.765,Z 681.922,A -85,B 0,C 180,E1 -7994.538,E2 -7994.538} C_VEL
LIN {X 0,Y 463.38,Z 695.178,A -85,B 0,C 180,E1 -7994.919,E2 -7994.919} C_VEL
LIN {X 0,Y 462.921,Z 707.34,A -85,B 0,C 180,E1 -7995.438,E2 -7995.438} C_VEL
LIN {X 0,Y 462.4,Z 719.622,A -85,B 0,C 180,E1 -7996.151,E2 -7996.151} C_VEL
LIN {X 0,Y 461.838,Z 730.804,A -85,B 0,C 180,E1 -7996.994,E2 -7996.994} C_VEL
LIN {X 0,Y 461.339,Z 741.664,A -85,B 0,C 180,E1 -7998.021,E2 -7998.021} C_VEL
LIN {X 0,Y 460.819,Z 750.204,A -85,B 0,C 180,E1 -7999.011,E2 -7999.011} C_VEL
LIN {X 0,Y 460.461,Z 758.086,A -85,B 0,C 180,E1 -8000.114,E2 -8000.114} C_VEL
LIN {X 0,Y 460.064,Z 765.784,A -85,B 0,C 180,E1 -8001.435,E2 -8001.435} C_VEL
LIN {X 0,Y 459.778,Z 772.88,A -85,B 0,C 180,E1 -8002.977,E2 -8002.977} C_VEL
LIN {X 0,Y 459.68,Z 777.604,A -85,B 0,C 180,E1 -8004.297,E2 -8004.297} C_VEL
LIN {X 0,Y 459.569,Z 781.215,A -85,B 0,C 180,E1 -8005.616,E2 -8005.616} C_VEL
LIN {X 0,Y 459.586,Z 783.079,A -85,B 0,C 180,E1 -8006.494,E2 -8006.494} C_VEL
LIN {X 0,Y 459.584,Z 784.475,A -85,B 0,C 180,E1 -8007.371,E2 -8007.371} C_VEL
LIN {X 0,Y 459.521,Z 786.075,A -85,B 0,C 180,E1 -8009.124,E2 -8009.124} C_VEL
LIN {X 0,Y 459.53,Z 786.291,A -85,B 0,C 180,E1 -8010.001,E2 -8010.001} C_VEL
LIN {X 0,Y 459.521,Z 786.074,A -85,B 0,C 180,E1 -8010.877,E2 -8010.877} C_VEL
LIN {X 0,Y 459.584,Z 784.47,A -85,B 0,C 180,E1 -8012.63,E2 -8012.63} C_VEL
LIN {X 0,Y 459.586,Z 783.072,A -85,B 0,C 180,E1 -8013.508,E2 -8013.508} C_VEL
LIN {X 0,Y 459.623,Z 780.138,A -85,B 0,C 180,E1 -8014.825,E2 -8014.825} C_VEL
LIN {X 0,Y 459.715,Z 775.135,A -85,B 0,C 180,E1 -8016.432,E2 -8016.432} C_VEL
LIN {X 0,Y 459.952,Z 769.039,A -85,B 0,C 180,E1 -8017.905,E2 -8017.905} C_VEL
LIN {X 0,Y 460.242,Z 762.137,A -85,B 0,C 180,E1 -8019.227,E2 -8019.227} C_VEL
LIN {X 0,Y 460.577,Z 755.089,A -85,B 0,C 180,E1 -8020.329,E2 -8020.329} C_VEL
LIN {X 0,Y 461.031,Z 746.599,A -85,B 0,C 180,E1 -8021.431,E2 -8021.431} C_VEL
LIN {X 0,Y 461.615,Z 736.653,A -85,B 0,C 180,E1 -8022.479,E2 -8022.479} C_VEL
LIN {X 0,Y 462.028,Z 725.726,A -85,B 0,C 180,E1 -8023.414,E2 -8023.414} C_VEL
LIN {X 0,Y 462.588,Z 714.355,A -85,B 0,C 180,E1 -8024.182,E2 -8024.182} C_VEL
LIN {X 0,Y 463.108,Z 702.693,A -85,B 0,C 180,E1 -8024.783,E2 -8024.783} C_VEL
LIN {X 0,Y 463.556,Z 689.24,A -85,B 0,C 180,E1 -8025.274,E2 -8025.274} C_VEL
LIN {X 0,Y 463.862,Z 675.931,A -85,B 0,C 180,E1 -8025.573,E2 -8025.573} C_VEL
LIN {X 0,Y 464.327,Z 592.04,A -85,B 0,C 180,E1 -8026.88,E2 -8026.88} C_VEL
LIN {X 0,Y 461.471,Z 574.126,A -85,B 0,C 180,E1 -8027.288,E2 -8027.288} C_VEL
LIN {X 0,Y 461.504,Z 571.285,A -85,B 0,C 180,E1 -8027.733,E2 -8027.733} C_VEL
LIN {X 0,Y 462.36,Z 553.644,A -85,B 0,C 180,E1 -8030.929,E2 -8030.929} C_VEL
LIN {X 0,Y 462.949,Z 540.969,A -85,B 0,C 180,E1 -8033.248,E2 -8033.248} C_VEL
LIN {X 0,Y 462.322,Z 535.878,A -85,B 0,C 180,E1 -8034.233,E2 -8034.233} C_VEL
LIN {X 0,Y 460.638,Z 527.263,A -85,B 0,C 180,E1 -8035.992,E2 -8035.992} C_VEL
LIN {X 0,Y 460.543,Z 527.103,A -85,B 0,C 180,E1 -8039.231,E2 -8039.231} C_VEL
LIN {X 0,Y 460.535,Z 527.121,A -85,B 0,C 180,E1 -8042.285,E2 -8042.285} C_VEL
LIN {X 0,Y 460.514,Z 527.118,A -85,B 0,C 180,E1 -8045.446,E2 -8045.446} C_VEL
LIN {X 0,Y 460.548,Z 527.116,A -85,B 0,C 180,E1 -8048.898,E2 -8048.898} C_VEL
LIN {X 0,Y 460.526,Z 527.121,A -85,B 0,C 180,E1 -8052.182,E2 -8052.182} C_VEL
LIN {X 0,Y 460.517,Z 527.12,A -85,B 0,C 180,E1 -8055.411,E2 -8055.411} C_VEL
LIN {X 0,Y 460.535,Z 527.122,A -85,B 0,C 180,E1 -8058.398,E2 -8058.398} C_VEL
LIN {X 0,Y 460.53,Z 527.117,A -85,B 0,C 180,E1 -8061.267,E2 -8061.267} C_VEL
LIN {X 0,Y 460.516,Z 527.122,A -85,B 0,C 180,E1 -8064.555,E2 -8064.555} C_VEL
LIN {X 0,Y 460.535,Z 527.12,A -85,B 0,C 180,E1 -8067.716,E2 -8067.716} C_VEL
LIN {X 0,Y 460.543,Z 527.12,A -85,B 0,C 180,E1 -8070.769,E2 -8070.769} C_VEL
LIN {X 0,Y 460.664,Z 527.302,A -85,B 0,C 180,E1 -8072.885,E2 -8072.885} C_VEL
LIN {X 0,Y 463.043,Z 539.435,A -85,B 0,C 180,E1 -8074.851,E2 -8074.851} C_VEL
LIN {X 0,Y 462.797,Z 553.765,A -85,B 0,C 180,E1 -8076.981,E2 -8076.981} C_VEL
LIN {X 0,Y 462.229,Z 573.928,A -85,B 0,C 180,E1 -8079.995,E2 -8079.995} C_VEL
LIN {X 0,Y 461.651,Z 593.641,A -85,B 0,C 180,E1 -8082.959,E2 -8082.959} C_VEL
LIN {X 0,Y 461.226,Z 610.035,A -85,B 0,C 180,E1 -8085.438,E2 -8085.438} C_VEL
LIN {X 0,Y 461.097,Z 616.764,A -85,B 0,C 180,E1 -8086.425,E2 -8086.425} C_VEL
LIN {X 0,Y 462.612,Z 630.283,A -85,B 0,C 180,E1 -8086.742,E2 -8086.742} C_VEL
LIN {X 0,Y 462.017,Z 696.592,A -85,B 0,C 180,E1 -8087.927,E2 -8087.927} C_VEL
LIN {X 0,Y 461.763,Z 706.463,A -85,B 0,C 180,E1 -8088.227,E2 -8088.227} C_VEL
LIN {X 0,Y 461.568,Z 715.885,A -85,B 0,C 180,E1 -8088.639,E2 -8088.639} C_VEL
LIN {X 0,Y 461.296,Z 726.236,A -85,B 0,C 180,E1 -8089.244,E2 -8089.244} C_VEL
LIN {X 0,Y 460.935,Z 736.181,A -85,B 0,C 180,E1 -8090.012,E2 -8090.012} C_VEL
LIN {X 0,Y 460.63,Z 744.042,A -85,B 0,C 180,E1 -8090.781,E2 -8090.781} C_VEL
LIN {X 0,Y 460.291,Z 751.412,A -85,B 0,C 180,E1 -8091.66,E2 -8091.66} C_VEL
LIN {X 0,Y 460.077,Z 757.492,A -85,B 0,C 180,E1 -8092.539,E2 -8092.539} C_VEL
LIN {X 0,Y 459.955,Z 763.323,A -85,B 0,C 180,E1 -8093.569,E2 -8093.569} C_VEL
LIN {X 0,Y 459.768,Z 768.613,A -85,B 0,C 180,E1 -8094.738,E2 -8094.738} C_VEL
LIN {X 0,Y 459.691,Z 772.973,A -85,B 0,C 180,E1 -8096.055,E2 -8096.055} C_VEL
LIN {X 0,Y 459.594,Z 775.988,A -85,B 0,C 180,E1 -8097.371,E2 -8097.371} C_VEL
LIN {X 0,Y 459.52,Z 777.329,A -85,B 0,C 180,E1 -8098.247,E2 -8098.247} C_VEL
LIN {X 0,Y 459.493,Z 778.166,A -85,B 0,C 180,E1 -8099.124,E2 -8099.124} C_VEL
LIN {X 0,Y 459.5,Z 778.468,A -85,B 0,C 180,E1 -8100,E2 -8100} C_VEL
LIN {X 0,Y 459.494,Z 778.183,A -85,B 0,C 180,E1 -8100.876,E2 -8100.876} C_VEL
LIN {X 0,Y 459.521,Z 777.393,A -85,B 0,C 180,E1 -8101.753,E2 -8101.753} C_VEL
LIN {X 0,Y 459.594,Z 776.099,A -85,B 0,C 180,E1 -8102.629,E2 -8102.629} C_VEL
LIN {X 0,Y 459.67,Z 773.131,A -85,B 0,C 180,E1 -8103.945,E2 -8103.945} C_VEL
LIN {X 0,Y 459.76,Z 768.857,A -85,B 0,C 180,E1 -8105.262,E2 -8105.262} C_VEL
LIN {X 0,Y 459.898,Z 763.993,A -85,B 0,C 180,E1 -8106.371,E2 -8106.371} C_VEL
LIN {X 0,Y 460.069,Z 757.931,A -85,B 0,C 180,E1 -8107.461,E2 -8107.461} C_VEL
LIN {X 0,Y 460.286,Z 751.95,A -85,B 0,C 180,E1 -8108.34,E2 -8108.34} C_VEL
LIN {X 0,Y 460.592,Z 744.698,A -85,B 0,C 180,E1 -8109.219,E2 -8109.219} C_VEL
LIN {X 0,Y 460.97,Z 735.792,A -85,B 0,C 180,E1 -8110.098,E2 -8110.098} C_VEL
LIN {X 0,Y 461.301,Z 725.68,A -85,B 0,C 180,E1 -8110.867,E2 -8110.867} C_VEL
LIN {X 0,Y 461.549,Z 716.272,A -85,B 0,C 180,E1 -8111.417,E2 -8111.417} C_VEL
LIN {X 0,Y 461.771,Z 706.964,A -85,B 0,C 180,E1 -8111.829,E2 -8111.829} C_VEL
LIN {X 0,Y 461.935,Z 697.291,A -85,B 0,C 180,E1 -8112.131,E2 -8112.131} C_VEL
LIN {X 0,Y 462.246,Z 670.194,A -85,B 0,C 180,E1 -8112.613,E2 -8112.613} C_VEL
LIN {X 0,Y 462.493,Z 628.864,A -85,B 0,C 180,E1 -8113.329,E2 -8113.329} C_VEL
LIN {X 0,Y 461.001,Z 616.658,A -85,B 0,C 180,E1 -8113.598,E2 -8113.598} C_VEL
LIN {X 0,Y 461.526,Z 598.39,A -85,B 0,C 180,E1 -8116.392,E2 -8116.392} C_VEL
LIN {X 0,Y 462.285,Z 575.004,A -85,B 0,C 180,E1 -8120.003,E2 -8120.003} C_VEL
LIN {X 0,Y 462.934,Z 555.598,A -85,B 0,C 180,E1 -8123.012,E2 -8123.012} C_VEL
LIN {X 0,Y 463.372,Z 541.967,A -85,B 0,C 180,E1 -8125.13,E2 -8125.13} C_VEL
LIN {X 0,Y 461.793,Z 532.906,A -85,B 0,C 180,E1 -8126.628,E2 -8126.628} C_VEL
LIN {X 0,Y 460.619,Z 527.216,A -85,B 0,C 180,E1 -8127.618,E2 -8127.618} C_VEL
LIN {X 0,Y 460.541,Z 527.12,A -85,B 0,C 180,E1 -8131.255,E2 -8131.255} C_VEL
LIN {X 0,Y 460.536,Z 527.116,A -85,B 0,C 180,E1 -8134.506,E2 -8134.506} C_VEL
LIN {X 0,Y 460.531,Z 527.121,A -85,B 0,C 180,E1 -8137.62,E2 -8137.62} C_VEL
LIN {X 0,Y 460.545,Z 527.103,A -85,B 0,C 180,E1 -8140.269,E2 -8140.269} C_VEL
LIN {X 0,Y 460.512,Z 527.101,A -85,B 0,C 180,E1 -8143.374,E2 -8143.374} C_VEL
LIN {X 0,Y 460.503,Z 527.12,A -85,B 0,C 180,E1 -8146.624,E2 -8146.624} C_VEL
LIN {X 0,Y 460.542,Z 527.098,A -85,B 0,C 180,E1 -8149.731,E2 -8149.731} C_VEL
LIN {X 0,Y 460.503,Z 527.118,A -85,B 0,C 180,E1 -8152.524,E2 -8152.524} C_VEL
LIN {X 0,Y 460.541,Z 527.114,A -85,B 0,C 180,E1 -8155.623,E2 -8155.623} C_VEL
LIN {X 0,Y 460.54,Z 527.117,A -85,B 0,C 180,E1 -8158.761,E2 -8158.761} C_VEL
LIN {X 0,Y 460.586,Z 527.111,A -85,B 0,C 180,E1 -8162.253,E2 -8162.253} C_VEL
LIN {X 0,Y 460.576,Z 527.115,A -85,B 0,C 180,E1 -8162.571,E2 -8162.571} C_VEL
LIN {X 0,Y 459.913,Z 527.202,A -85,B 0,C 180,E1 -8163.301,E2 -8163.301} C_VEL
LIN {X 0,Y 457.061,Z 527.554,A -85,B 0,C 180,E1 -8164.486,E2 -8164.486} C_VEL
LIN {X 0,Y 454.638,Z 527.849,A -85,B 0,C 180,E1 -8165.441,E2 -8165.441} C_VEL
LIN {X 0,Y 453.586,Z 527.977,A -85,B 0,C 180,E1 -8166.179,E2 -8166.179} C_VEL
LIN {X 0,Y 453.494,Z 527.989,A -85,B 0,C 180,E1 -8166.43,E2 -8166.43} C_VEL
LIN {X 0,Y 453.526,Z 528.096,A -85,B 0,C 180,E1 -8167.627,E2 -8167.627} C_VEL
LIN {X 0,Y 455.114,Z 536.539,A -85,B 0,C 180,E1 -8169.668,E2 -8169.668} C_VEL
LIN {X 0,Y 454.612,Z 549.472,A -85,B 0,C 180,E1 -8172.465,E2 -8172.465} C_VEL
LIN {X 0,Y 455.204,Z 552.74,A -85,B 0,C 180,E1 -8172.591,E2 -8172.591} C_VEL
LIN {X 0,Y 457.819,Z 567.131,A -85,B 0,C 180,E1 -8172.927,E2 -8172.927} C_VEL
LIN {X 0,Y 457.018,Z 656.718,A -85,B 0,C 180,E1 -8174.359,E2 -8174.359} C_VEL
LIN {X 0,Y 456.66,Z 670.593,A -85,B 0,C 180,E1 -8174.775,E2 -8174.775} C_VEL
LIN {X 0,Y 456.212,Z 682.998,A -85,B 0,C 180,E1 -8175.331,E2 -8175.331} C_VEL
LIN {X 0,Y 455.71,Z 694.847,A -85,B 0,C 180,E1 -8176.056,E2 -8176.056} C_VEL
LIN {X 0,Y 455.187,Z 706.334,A -85,B 0,C 180,E1 -8176.96,E2 -8176.96} C_VEL
LIN {X 0,Y 454.617,Z 716.45,A -85,B 0,C 180,E1 -8177.953,E2 -8177.953} C_VEL
LIN {X 0,Y 454.084,Z 725.636,A -85,B 0,C 180,E1 -8179.07,E2 -8179.07} C_VEL
LIN {X 0,Y 453.573,Z 734.554,A -85,B 0,C 180,E1 -8180.411,E2 -8180.411} C_VEL
LIN {X 0,Y 453.177,Z 741.732,A -85,B 0,C 180,E1 -8181.752,E2 -8181.752} C_VEL
LIN {X 0,Y 452.885,Z 746.576,A -85,B 0,C 180,E1 -8182.868,E2 -8182.868} C_VEL
LIN {X 0,Y 452.826,Z 751.277,A -85,B 0,C 180,E1 -8184.209,E2 -8184.209} C_VEL
LIN {X 0,Y 452.585,Z 754.879,A -85,B 0,C 180,E1 -8185.546,E2 -8185.546} C_VEL
LIN {X 0,Y 452.622,Z 756.736,A -85,B 0,C 180,E1 -8186.438,E2 -8186.438} C_VEL
LIN {X 0,Y 452.535,Z 758.141,A -85,B 0,C 180,E1 -8187.329,E2 -8187.329} C_VEL
LIN {X 0,Y 452.431,Z 759.758,A -85,B 0,C 180,E1 -8189.109,E2 -8189.109} C_VEL
LIN {X 0,Y 452.435,Z 759.993,A -85,B 0,C 180,E1 -8189.999,E2 -8189.999} C_VEL
LIN {X 0,Y 452.43,Z 759.808,A -85,B 0,C 180,E1 -8190.889,E2 -8190.889} C_VEL
LIN {X 0,Y 452.534,Z 758.26,A -85,B 0,C 180,E1 -8192.67,E2 -8192.67} C_VEL
LIN {X 0,Y 452.606,Z 756.906,A -85,B 0,C 180,E1 -8193.56,E2 -8193.56} C_VEL
LIN {X 0,Y 452.602,Z 754.043,A -85,B 0,C 180,E1 -8194.898,E2 -8194.898} C_VEL
LIN {X 0,Y 452.845,Z 750.155,A -85,B 0,C 180,E1 -8196.236,E2 -8196.236} C_VEL
LIN {X 0,Y 452.988,Z 745.149,A -85,B 0,C 180,E1 -8197.577,E2 -8197.577} C_VEL
LIN {X 0,Y 453.36,Z 738.843,A -85,B 0,C 180,E1 -8198.917,E2 -8198.917} C_VEL
LIN {X 0,Y 453.756,Z 730.946,A -85,B 0,C 180,E1 -8200.259,E2 -8200.259} C_VEL
LIN {X 0,Y 454.3,Z 721.122,A -85,B 0,C 180,E1 -8201.601,E2 -8201.601} C_VEL
LIN {X 0,Y 454.987,Z 710.98,A -85,B 0,C 180,E1 -8202.698,E2 -8202.698} C_VEL
LIN {X 0,Y 455.432,Z 700.053,A -85,B 0,C 180,E1 -8203.654,E2 -8203.654} C_VEL
LIN {X 0,Y 455.984,Z 689.425,A -85,B 0,C 180,E1 -8204.39,E2 -8204.39} C_VEL
LIN {X 0,Y 456.436,Z 678.085,A -85,B 0,C 180,E1 -8205.002,E2 -8205.002} C_VEL
LIN {X 0,Y 456.839,Z 665.177,A -85,B 0,C 180,E1 -8205.503,E2 -8205.503} C_VEL
LIN {X 0,Y 457.117,Z 651.399,A -85,B 0,C 180,E1 -8205.836,E2 -8205.836} C_VEL
LIN {X 0,Y 457.738,Z 565.848,A -85,B 0,C 180,E1 -8207.19,E2 -8207.19} C_VEL
LIN {X 0,Y 454.643,Z 549.953,A -85,B 0,C 180,E1 -8207.589,E2 -8207.589} C_VEL
LIN {X 0,Y 454.617,Z 548.486,A -85,B 0,C 180,E1 -8207.8,E2 -8207.8} C_VEL
LIN {X 0,Y 455.141,Z 536.963,A -85,B 0,C 180,E1 -8210.329,E2 -8210.329} C_VEL
LIN {X 0,Y 453.532,Z 528.05,A -85,B 0,C 180,E1 -8212.491,E2 -8212.491} C_VEL
LIN {X 0,Y 453.517,Z 527.987,A -85,B 0,C 180,E1 -8215.998,E2 -8215.998} C_VEL
LIN {X 0,Y 453.51,Z 527.99,A -85,B 0,C 180,E1 -8218.711,E2 -8218.711} C_VEL
LIN {X 0,Y 453.464,Z 527.999,A -85,B 0,C 180,E1 -8221.798,E2 -8221.798} C_VEL
LIN {X 0,Y 453.48,Z 527.998,A -85,B 0,C 180,E1 -8224.988,E2 -8224.988} C_VEL
LIN {X 0,Y 453.471,Z 527.995,A -85,B 0,C 180,E1 -8228.31,E2 -8228.31} C_VEL
LIN {X 0,Y 453.491,Z 527.989,A -85,B 0,C 180,E1 -8230.608,E2 -8230.608} C_VEL
LIN {X 0,Y 453.46,Z 528.002,A -85,B 0,C 180,E1 -8233.244,E2 -8233.244} C_VEL
LIN {X 0,Y 453.462,Z 527.997,A -85,B 0,C 180,E1 -8235.778,E2 -8235.778} C_VEL
LIN {X 0,Y 453.511,Z 527.992,A -85,B 0,C 180,E1 -8239.405,E2 -8239.405} C_VEL
LIN {X 0,Y 453.473,Z 527.987,A -85,B 0,C 180,E1 -8242.222,E2 -8242.222} C_VEL
LIN {X 0,Y 453.497,Z 527.996,A -85,B 0,C 180,E1 -8245.219,E2 -8245.219} C_VEL
LIN {X 0,Y 453.463,Z 527.994,A -85,B 0,C 180,E1 -8248.473,E2 -8248.473} C_VEL
LIN {X 0,Y 453.51,Z 527.995,A -85,B 0,C 180,E1 -8251.288,E2 -8251.288} C_VEL
LIN {X 0,Y 453.519,Z 527.989,A -85,B 0,C 180,E1 -8254.284,E2 -8254.284} C_VEL
LIN {X 0,Y 453.473,Z 527.997,A -85,B 0,C 180,E1 -8257.204,E2 -8257.204} C_VEL
LIN {X 0,Y 453.498,Z 527.992,A -85,B 0,C 180,E1 -8260.066,E2 -8260.066} C_VEL
LIN {X 0,Y 453.5,Z 527.989,A -85,B 0,C 180,E1 -8262.875,E2 -8262.875} C_VEL
LIN {X 0,Y 453.506,Z 527.996,A -85,B 0,C 180,E1 -8265.644,E2 -8265.644} C_VEL
LIN {X 0,Y 453.552,Z 527.982,A -85,B 0,C 180,E1 -8268.379,E2 -8268.379} C_VEL
LIN {X 0,Y 453.644,Z 527.975,A -85,B 0,C 180,E1 -8271.985,E2 -8271.985} C_VEL
LIN {X 0,Y 453.665,Z 527.97,A -85,B 0,C 180,E1 -8274.667,E2 -8274.667} C_VEL
LIN {X 0,Y 453.758,Z 527.956,A -85,B 0,C 180,E1 -8277.337,E2 -8277.337} C_VEL
LIN {X 0,Y 453.817,Z 527.954,A -85,B 0,C 180,E1 -8280,E2 -8280} C_VEL
LIN {X 0,Y 453.759,Z 527.955,A -85,B 0,C 180,E1 -8282.663,E2 -8282.663} C_VEL
LIN {X 0,Y 453.67,Z 527.971,A -85,B 0,C 180,E1 -8286.225,E2 -8286.225} C_VEL
LIN {X 0,Y 453.585,Z 527.979,A -85,B 0,C 180,E1 -8288.914,E2 -8288.914} C_VEL
LIN {X 0,Y 453.594,Z 527.979,A -85,B 0,C 180,E1 -8292.551,E2 -8292.551} C_VEL
LIN {X 0,Y 453.537,Z 527.983,A -85,B 0,C 180,E1 -8296.196,E2 -8296.196} C_VEL
LIN {X 0,Y 453.513,Z 527.991,A -85,B 0,C 180,E1 -8299.041,E2 -8299.041} C_VEL
LIN {X 0,Y 453.469,Z 527.997,A -85,B 0,C 180,E1 -8301.837,E2 -8301.837} C_VEL
LIN {X 0,Y 453.507,Z 527.99,A -85,B 0,C 180,E1 -8304.735,E2 -8304.735} C_VEL
LIN {X 0,Y 453.531,Z 527.991,A -85,B 0,C 180,E1 -8307.962,E2 -8307.962} C_VEL
LIN {X 0,Y 453.46,Z 527.999,A -85,B 0,C 180,E1 -8311.526,E2 -8311.526} C_VEL
LIN {X 0,Y 453.483,Z 527.991,A -85,B 0,C 180,E1 -8314.778,E2 -8314.778} C_VEL
LIN {X 0,Y 453.468,Z 527.995,A -85,B 0,C 180,E1 -8318.311,E2 -8318.311} C_VEL
LIN {X 0,Y 453.488,Z 527.992,A -85,B 0,C 180,E1 -8320.61,E2 -8320.61} C_VEL
LIN {X 0,Y 453.45,Z 527.993,A -85,B 0,C 180,E1 -8323.245,E2 -8323.245} C_VEL
LIN {X 0,Y 453.473,Z 527.998,A -85,B 0,C 180,E1 -8325.781,E2 -8325.781} C_VEL
LIN {X 0,Y 453.493,Z 527.995,A -85,B 0,C 180,E1 -8328.212,E2 -8328.212} C_VEL
LIN {X 0,Y 453.527,Z 527.984,A -85,B 0,C 180,E1 -8330.789,E2 -8330.789} C_VEL
LIN {X 0,Y 453.454,Z 527.999,A -85,B 0,C 180,E1 -8333.918,E2 -8333.918} C_VEL
LIN {X 0,Y 453.48,Z 527.976,A -85,B 0,C 180,E1 -8337.152,E2 -8337.152} C_VEL
LIN {X 0,Y 453.473,Z 527.971,A -85,B 0,C 180,E1 -8340.269,E2 -8340.269} C_VEL
LIN {X 0,Y 453.516,Z 527.97,A -85,B 0,C 180,E1 -8343.296,E2 -8343.296} C_VEL
LIN {X 0,Y 453.581,Z 528.15,A -85,B 0,C 180,E1 -8343.784,E2 -8343.784} C_VEL
LIN {X 0,Y 455.675,Z 538.872,A -85,B 0,C 180,E1 -8345.991,E2 -8345.991} C_VEL
LIN {X 0,Y 456.008,Z 543.351,A -85,B 0,C 180,E1 -8346.859,E2 -8346.859} C_VEL
LIN {X 0,Y 455.073,Z 559.787,A -85,B 0,C 180,E1 -8349.903,E2 -8349.903} C_VEL
LIN {X 0,Y 454.483,Z 573.517,A -85,B 0,C 180,E1 -8352.404,E2 -8352.404} C_VEL
LIN {X 0,Y 455.244,Z 578.547,A -85,B 0,C 180,E1 -8352.557,E2 -8352.557} C_VEL
LIN {X 0,Y 457.676,Z 594.661,A -85,B 0,C 180,E1 -8352.911,E2 -8352.911} C_VEL
LIN {X 0,Y 456.939,Z 681.727,A -85,B 0,C 180,E1 -8354.301,E2 -8354.301} C_VEL
LIN {X 0,Y 456.505,Z 694.979,A -85,B 0,C 180,E1 -8354.686,E2 -8354.686} C_VEL
LIN {X 0,Y 456.024,Z 707.14,A -85,B 0,C 180,E1 -8355.212,E2 -8355.212} C_VEL
LIN {X 0,Y 455.485,Z 719.42,A -85,B 0,C 180,E1 -8355.936,E2 -8355.936} C_VEL
LIN {X 0,Y 454.858,Z 731.479,A -85,B 0,C 180,E1 -8356.868,E2 -8356.868} C_VEL
LIN {X 0,Y 454.314,Z 742.506,A -85,B 0,C 180,E1 -8357.947,E2 -8357.947} C_VEL
LIN {X 0,Y 453.724,Z 751.679,A -85,B 0,C 180,E1 -8359.063,E2 -8359.063} C_VEL
LIN {X 0,Y 453.257,Z 760.62,A -85,B 0,C 180,E1 -8360.406,E2 -8360.406} C_VEL
LIN {X 0,Y 452.937,Z 767.819,A -85,B 0,C 180,E1 -8361.749,E2 -8361.749} C_VEL
LIN {X 0,Y 452.723,Z 772.676,A -85,B 0,C 180,E1 -8362.867,E2 -8362.867} C_VEL
LIN {X 0,Y 452.583,Z 777.399,A -85,B 0,C 180,E1 -8364.208,E2 -8364.208} C_VEL
LIN {X 0,Y 452.491,Z 781.011,A -85,B 0,C 180,E1 -8365.547,E2 -8365.547} C_VEL
LIN {X 0,Y 452.482,Z 782.874,A -85,B 0,C 180,E1 -8366.439,E2 -8366.439} C_VEL
LIN {X 0,Y 452.508,Z 784.271,A -85,B 0,C 180,E1 -8367.33,E2 -8367.33} C_VEL
LIN {X 0,Y 452.428,Z 785.871,A -85,B 0,C 180,E1 -8369.111,E2 -8369.111} C_VEL
LIN {X 0,Y 452.434,Z 786.086,A -85,B 0,C 180,E1 -8370.001,E2 -8370.001} C_VEL
LIN {X 0,Y 452.428,Z 785.869,A -85,B 0,C 180,E1 -8370.891,E2 -8370.891} C_VEL
LIN {X 0,Y 452.508,Z 784.265,A -85,B 0,C 180,E1 -8372.671,E2 -8372.671} C_VEL
LIN {X 0,Y 452.483,Z 782.867,A -85,B 0,C 180,E1 -8373.563,E2 -8373.563} C_VEL
LIN {X 0,Y 452.552,Z 779.933,A -85,B 0,C 180,E1 -8374.901,E2 -8374.901} C_VEL
LIN {X 0,Y 452.629,Z 775.349,A -85,B 0,C 180,E1 -8376.417,E2 -8376.417} C_VEL
LIN {X 0,Y 452.894,Z 768.833,A -85,B 0,C 180,E1 -8378.029,E2 -8378.029} C_VEL
LIN {X 0,Y 453.211,Z 761.93,A -85,B 0,C 180,E1 -8379.372,E2 -8379.372} C_VEL
LIN {X 0,Y 453.624,Z 753.293,A -85,B 0,C 180,E1 -8380.715,E2 -8380.715} C_VEL
LIN {X 0,Y 454.171,Z 744.441,A -85,B 0,C 180,E1 -8381.832,E2 -8381.832} C_VEL
LIN {X 0,Y 454.694,Z 733.833,A -85,B 0,C 180,E1 -8382.924,E2 -8382.924} C_VEL
LIN {X 0,Y 455.273,Z 722.546,A -85,B 0,C 180,E1 -8383.844,E2 -8383.844} C_VEL
LIN {X 0,Y 455.872,Z 710.232,A -85,B 0,C 180,E1 -8384.623,E2 -8384.623} C_VEL
LIN {X 0,Y 456.424,Z 697.197,A -85,B 0,C 180,E1 -8385.233,E2 -8385.233} C_VEL
LIN {X 0,Y 456.909,Z 683.889,A -85,B 0,C 180,E1 -8385.645,E2 -8385.645} C_VEL
LIN {X 0,Y 457.138,Z 661.397,A -85,B 0,C 180,E1 -8386.037,E2 -8386.037} C_VEL
LIN {X 0,Y 457.562,Z 593.046,A -85,B 0,C 180,E1 -8387.117,E2 -8387.117} C_VEL
LIN {X 0,Y 454.495,Z 573.909,A -85,B 0,C 180,E1 -8387.562,E2 -8387.562} C_VEL
LIN {X 0,Y 454.546,Z 571.084,A -85,B 0,C 180,E1 -8388.014,E2 -8388.014} C_VEL
LIN {X 0,Y 455.383,Z 554.714,A -85,B 0,C 180,E1 -8391.028,E2 -8391.028} C_VEL
LIN {X 0,Y 456.025,Z 542.054,A -85,B 0,C 180,E1 -8393.382,E2 -8393.382} C_VEL
LIN {X 0,Y 454.853,Z 534.418,A -85,B 0,C 180,E1 -8394.901,E2 -8394.901} C_VEL
LIN {X 0,Y 453.587,Z 528.148,A -85,B 0,C 180,E1 -8396.217,E2 -8396.217} C_VEL
LIN {X 0,Y 453.513,Z 527.977,A -85,B 0,C 180,E1 -8398.712,E2 -8398.712} C_VEL
LIN {X 0,Y 453.468,Z 528,A -85,B 0,C 180,E1 -8401.8,E2 -8401.8} C_VEL
LIN {X 0,Y 453.484,Z 527.994,A -85,B 0,C 180,E1 -8404.99,E2 -8404.99} C_VEL
LIN {X 0,Y 453.468,Z 528,A -85,B 0,C 180,E1 -8408.312,E2 -8408.312} C_VEL
LIN {X 0,Y 453.498,Z 527.995,A -85,B 0,C 180,E1 -8410.609,E2 -8410.609} C_VEL
LIN {X 0,Y 453.458,Z 527.999,A -85,B 0,C 180,E1 -8413.244,E2 -8413.244} C_VEL
LIN {X 0,Y 453.467,Z 528,A -85,B 0,C 180,E1 -8415.779,E2 -8415.779} C_VEL
LIN {X 0,Y 453.482,Z 527.999,A -85,B 0,C 180,E1 -8418.209,E2 -8418.209} C_VEL
LIN {X 0,Y 453.519,Z 527.992,A -85,B 0,C 180,E1 -8420.79,E2 -8420.79} C_VEL
LIN {X 0,Y 453.46,Z 528.001,A -85,B 0,C 180,E1 -8423.918,E2 -8423.918} C_VEL
LIN {X 0,Y 453.486,Z 527.996,A -85,B 0,C 180,E1 -8427.151,E2 -8427.151} C_VEL
LIN {X 0,Y 453.478,Z 528.001,A -85,B 0,C 180,E1 -8430.268,E2 -8430.268} C_VEL
LIN {X 0,Y 453.627,Z 528.206,A -85,B 0,C 180,E1 -8432.601,E2 -8432.601} C_VEL
LIN {X 0,Y 455.922,Z 539.255,A -85,B 0,C 180,E1 -8434.43,E2 -8434.43} C_VEL
LIN {X 0,Y 456.277,Z 544.103,A -85,B 0,C 180,E1 -8435.183,E2 -8435.183} C_VEL
LIN {X 0,Y 455.664,Z 564.619,A -85,B 0,C 180,E1 -8438.274,E2 -8438.274} C_VEL
LIN {X 0,Y 454.957,Z 586.143,A -85,B 0,C 180,E1 -8441.538,E2 -8441.538} C_VEL
LIN {X 0,Y 454.411,Z 607.263,A -85,B 0,C 180,E1 -8444.756,E2 -8444.756} C_VEL
LIN {X 0,Y 454.141,Z 616.854,A -85,B 0,C 180,E1 -8446.184,E2 -8446.184} C_VEL
LIN {X 0,Y 455.754,Z 630.506,A -85,B 0,C 180,E1 -8446.523,E2 -8446.523} C_VEL
LIN {X 0,Y 455.082,Z 696.739,A -85,B 0,C 180,E1 -8447.74,E2 -8447.74} C_VEL
LIN {X 0,Y 454.82,Z 707.275,A -85,B 0,C 180,E1 -8448.072,E2 -8448.072} C_VEL
LIN {X 0,Y 454.561,Z 717.055,A -85,B 0,C 180,E1 -8448.518,E2 -8448.518} C_VEL
LIN {X 0,Y 454.246,Z 727.958,A -85,B 0,C 180,E1 -8449.188,E2 -8449.188} C_VEL
LIN {X 0,Y 453.87,Z 737.436,A -85,B 0,C 180,E1 -8449.968,E2 -8449.968} C_VEL
LIN {X 0,Y 453.622,Z 744.123,A -85,B 0,C 180,E1 -8450.638,E2 -8450.638} C_VEL
LIN {X 0,Y 453.27,Z 751.485,A -85,B 0,C 180,E1 -8451.53,E2 -8451.53} C_VEL
LIN {X 0,Y 453.023,Z 757.556,A -85,B 0,C 180,E1 -8452.423,E2 -8452.423} C_VEL
LIN {X 0,Y 452.919,Z 762.33,A -85,B 0,C 180,E1 -8453.265,E2 -8453.265} C_VEL
LIN {X 0,Y 452.782,Z 766.782,A -85,B 0,C 180,E1 -8454.209,E2 -8454.209} C_VEL
LIN {X 0,Y 452.613,Z 770.233,A -85,B 0,C 180,E1 -8455.101,E2 -8455.101} C_VEL
LIN {X 0,Y 452.576,Z 774.177,A -85,B 0,C 180,E1 -8456.439,E2 -8456.439} C_VEL
LIN {X 0,Y 452.521,Z 776.048,A -85,B 0,C 180,E1 -8457.33,E2 -8457.33} C_VEL
LIN {X 0,Y 452.436,Z 777.39,A -85,B 0,C 180,E1 -8458.22,E2 -8458.22} C_VEL
LIN {X 0,Y 452.402,Z 778.223,A -85,B 0,C 180,E1 -8459.11,E2 -8459.11} C_VEL
LIN {X 0,Y 452.405,Z 778.524,A -85,B 0,C 180,E1 -8460,E2 -8460} C_VEL
LIN {X 0,Y 452.403,Z 778.233,A -85,B 0,C 180,E1 -8460.89,E2 -8460.89} C_VEL
LIN {X 0,Y 452.438,Z 777.431,A -85,B 0,C 180,E1 -8461.78,E2 -8461.78} C_VEL
LIN {X 0,Y 452.521,Z 776.123,A -85,B 0,C 180,E1 -8462.671,E2 -8462.671} C_VEL
LIN {X 0,Y 452.565,Z 773.133,A -85,B 0,C 180,E1 -8464.007,E2 -8464.007} C_VEL
LIN {X 0,Y 452.704,Z 768.827,A -85,B 0,C 180,E1 -8465.345,E2 -8465.345} C_VEL
LIN {X 0,Y 452.85,Z 762.941,A -85,B 0,C 180,E1 -8466.66,E2 -8466.66} C_VEL
LIN {X 0,Y 453.006,Z 757.822,A -85,B 0,C 180,E1 -8467.578,E2 -8467.578} C_VEL
LIN {X 0,Y 453.261,Z 751.801,A -85,B 0,C 180,E1 -8468.471,E2 -8468.471} C_VEL
LIN {X 0,Y 453.56,Z 744.502,A -85,B 0,C 180,E1 -8469.364,E2 -8469.364} C_VEL
LIN {X 0,Y 453.953,Z 735.538,A -85,B 0,C 180,E1 -8470.256,E2 -8470.256} C_VEL
LIN {X 0,Y 454.313,Z 725.288,A -85,B 0,C 180,E1 -8471.037,E2 -8471.037} C_VEL
LIN {X 0,Y 454.533,Z 716.865,A -85,B 0,C 180,E1 -8471.539,E2 -8471.539} C_VEL
LIN {X 0,Y 454.798,Z 707.026,A -85,B 0,C 180,E1 -8471.985,E2 -8471.985} C_VEL
LIN {X 0,Y 454.967,Z 697.386,A -85,B 0,C 180,E1 -8472.291,E2 -8472.291} C_VEL
LIN {X 0,Y 455.307,Z 668.69,A -85,B 0,C 180,E1 -8472.814,E2 -8472.814} C_VEL
LIN {X 0,Y 455.515,Z 629.077,A -85,B 0,C 180,E1 -8473.517,E2 -8473.517} C_VEL
LIN {X 0,Y 454.004,Z 616.505,A -85,B 0,C 180,E1 -8473.812,E2 -8473.812} C_VEL
LIN {X 0,Y 454.543,Z 597.665,A -85,B 0,C 180,E1 -8476.731,E2 -8476.731} C_VEL
LIN {X 0,Y 455.309,Z 576.117,A -85,B 0,C 180,E1 -8480.087,E2 -8480.087} C_VEL
LIN {X 0,Y 455.989,Z 556.59,A -85,B 0,C 180,E1 -8483.143,E2 -8483.143} C_VEL
LIN {X 0,Y 456.408,Z 542.881,A -85,B 0,C 180,E1 -8485.297,E2 -8485.297} C_VEL
LIN {X 0,Y 453.995,Z 530.206,A -85,B 0,C 180,E1 -8487.422,E2 -8487.422} C_VEL
LIN {X 0,Y 453.58,Z 528.078,A -85,B 0,C 180,E1 -8487.831,E2 -8487.831} C_VEL
LIN {X 0,Y 453.47,Z 528.002,A -85,B 0,C 180,E1 -8491.525,E2 -8491.525} C_VEL
LIN {X 0,Y 453.492,Z 527.994,A -85,B 0,C 180,E1 -8494.777,E2 -8494.777} C_VEL
LIN {X 0,Y 453.477,Z 527.993,A -85,B 0,C 180,E1 -8498.311,E2 -8498.311} C_VEL
LIN {X 0,Y 453.498,Z 527.981,A -85,B 0,C 180,E1 -8500.609,E2 -8500.609} C_VEL
LIN {X 0,Y 453.464,Z 527.989,A -85,B 0,C 180,E1 -8504.222,E2 -8504.222} C_VEL
LIN {X 0,Y 453.467,Z 528,A -85,B 0,C 180,E1 -8507.005,E2 -8507.005} C_VEL
LIN {X 0,Y 453.498,Z 527.979,A -85,B 0,C 180,E1 -8509.409,E2 -8509.409} C_VEL
LIN {X 0,Y 453.456,Z 527.998,A -85,B 0,C 180,E1 -8512.81,E2 -8512.81} C_VEL
LIN {X 0,Y 453.472,Z 527.993,A -85,B 0,C 180,E1 -8516.086,E2 -8516.086} C_VEL
LIN {X 0,Y 453.481,Z 527.998,A -85,B 0,C 180,E1 -8519.24,E2 -8519.24} C_VEL
LIN {X 0,Y 453.519,Z 527.991,A -85,B 0,C 180,E1 -8522.564,E2 -8522.564} C_VEL
LIN {X 0,Y 453.511,Z 527.987,A -85,B 0,C 180,E1 -8525.265,E2 -8525.265} C_VEL
LIN {X 0,Y 453.494,Z 527.989,A -85,B 0,C 180,E1 -8526.43,E2 -8526.43} C_VEL
LIN {X 0,Y 453.248,Z 528.312,A -85,B 0,C 180,E1 -8526.921,E2 -8526.921} C_VEL
LIN {X 0,Y 452.264,Z 529.762,A -85,B 0,C 180,E1 -8527.633,E2 -8527.633} C_VEL
LIN {X 0,Y 450.905,Z 532.027,A -85,B 0,C 180,E1 -8528.308,E2 -8528.308} C_VEL
LIN {X 0,Y 448.438,Z 537.935,A -85,B 0,C 180,E1 -8529.628,E2 -8529.628} C_VEL
LIN {X 0,Y 448.116,Z 539.979,A -85,B 0,C 180,E1 -8530.073,E2 -8530.073} C_VEL
LIN {X 0,Y 447.668,Z 549.675,A -85,B 0,C 180,E1 -8532.184,E2 -8532.184} C_VEL
LIN {X 0,Y 448.193,Z 552.582,A -85,B 0,C 180,E1 -8532.303,E2 -8532.303} C_VEL
LIN {X 0,Y 451.035,Z 567.249,A -85,B 0,C 180,E1 -8532.66,E2 -8532.66} C_VEL
LIN {X 0,Y 450.199,Z 656.94,A -85,B 0,C 180,E1 -8534.116,E2 -8534.116} C_VEL
LIN {X 0,Y 449.824,Z 670.81,A -85,B 0,C 180,E1 -8534.538,E2 -8534.538} C_VEL
LIN {X 0,Y 449.35,Z 683.211,A -85,B 0,C 180,E1 -8535.102,E2 -8535.102} C_VEL
LIN {X 0,Y 448.826,Z 695.058,A -85,B 0,C 180,E1 -8535.838,E2 -8535.838} C_VEL
LIN {X 0,Y 448.249,Z 707.098,A -85,B 0,C 180,E1 -8536.804,E2 -8536.804} C_VEL
LIN {X 0,Y 447.689,Z 716.659,A -85,B 0,C 180,E1 -8537.764,E2 -8537.764} C_VEL
LIN {X 0,Y 447.109,Z 725.845,A -85,B 0,C 180,E1 -8538.897,E2 -8538.897} C_VEL
LIN {X 0,Y 446.557,Z 734.762,A -85,B 0,C 180,E1 -8540.259,E2 -8540.259} C_VEL
LIN {X 0,Y 446.131,Z 741.939,A -85,B 0,C 180,E1 -8541.62,E2 -8541.62} C_VEL
LIN {X 0,Y 445.803,Z 747.872,A -85,B 0,C 180,E1 -8543.036,E2 -8543.036} C_VEL
LIN {X 0,Y 445.649,Z 752.799,A -85,B 0,C 180,E1 -8544.57,E2 -8544.57} C_VEL
LIN {X 0,Y 445.501,Z 755.085,A -85,B 0,C 180,E1 -8545.475,E2 -8545.475} C_VEL
LIN {X 0,Y 445.525,Z 756.942,A -85,B 0,C 180,E1 -8546.382,E2 -8546.382} C_VEL
LIN {X 0,Y 445.464,Z 758.346,A -85,B 0,C 180,E1 -8547.286,E2 -8547.286} C_VEL
LIN {X 0,Y 445.341,Z 759.962,A -85,B 0,C 180,E1 -8549.095,E2 -8549.095} C_VEL
LIN {X 0,Y 445.342,Z 760.198,A -85,B 0,C 180,E1 -8549.999,E2 -8549.999} C_VEL
LIN {X 0,Y 445.341,Z 760.012,A -85,B 0,C 180,E1 -8550.903,E2 -8550.903} C_VEL
LIN {X 0,Y 445.463,Z 758.464,A -85,B 0,C 180,E1 -8552.712,E2 -8552.712} C_VEL
LIN {X 0,Y 445.509,Z 757.11,A -85,B 0,C 180,E1 -8553.617,E2 -8553.617} C_VEL
LIN {X 0,Y 445.539,Z 754.247,A -85,B 0,C 180,E1 -8554.976,E2 -8554.976} C_VEL
LIN {X 0,Y 445.778,Z 750.359,A -85,B 0,C 180,E1 -8556.335,E2 -8556.335} C_VEL
LIN {X 0,Y 445.956,Z 745.352,A -85,B 0,C 180,E1 -8557.697,E2 -8557.697} C_VEL
LIN {X 0,Y 446.351,Z 739.045,A -85,B 0,C 180,E1 -8559.058,E2 -8559.058} C_VEL
LIN {X 0,Y 446.774,Z 731.148,A -85,B 0,C 180,E1 -8560.421,E2 -8560.421} C_VEL
LIN {X 0,Y 447.355,Z 721.323,A -85,B 0,C 180,E1 -8561.784,E2 -8561.784} C_VEL
LIN {X 0,Y 448.053,Z 711.311,A -85,B 0,C 180,E1 -8562.885,E2 -8562.885} C_VEL
LIN {X 0,Y 448.539,Z 699.936,A -85,B 0,C 180,E1 -8563.894,E2 -8563.894} C_VEL
LIN {X 0,Y 449.121,Z 689.622,A -85,B 0,C 180,E1 -8564.614,E2 -8564.614} C_VEL
LIN {X 0,Y 449.598,Z 678.28,A -85,B 0,C 180,E1 -8565.236,E2 -8565.236} C_VEL
LIN {X 0,Y 450.028,Z 665.366,A -85,B 0,C 180,E1 -8565.743,E2 -8565.743} C_VEL
LIN {X 0,Y 450.309,Z 651.579,A -85,B 0,C 180,E1 -8566.082,E2 -8566.082} C_VEL
LIN {X 0,Y 450.935,Z 566.445,A -85,B 0,C 180,E1 -8567.45,E2 -8567.45} C_VEL
LIN {X 0,Y 447.714,Z 549.967,A -85,B 0,C 180,E1 -8567.879,E2 -8567.879} C_VEL
LIN {X 0,Y 447.714,Z 547.728,A -85,B 0,C 180,E1 -8568.296,E2 -8568.296} C_VEL
LIN {X 0,Y 448.167,Z 538.2,A -85,B 0,C 180,E1 -8570.42,E2 -8570.42} C_VEL
LIN {X 0,Y 446.496,Z 528.963,A -85,B 0,C 180,E1 -8572.682,E2 -8572.682} C_VEL
LIN {X 0,Y 446.475,Z 528.864,A -85,B 0,C 180,E1 -8576.201,E2 -8576.201} C_VEL
LIN {X 0,Y 446.448,Z 528.865,A -85,B 0,C 180,E1 -8579.208,E2 -8579.208} C_VEL
LIN {X 0,Y 446.421,Z 528.873,A -85,B 0,C 180,E1 -8582.36,E2 -8582.36} C_VEL
LIN {X 0,Y 446.419,Z 528.874,A -85,B 0,C 180,E1 -8585.625,E2 -8585.625} C_VEL
LIN {X 0,Y 446.458,Z 528.872,A -85,B 0,C 180,E1 -8589.024,E2 -8589.024} C_VEL
LIN {X 0,Y 446.429,Z 528.873,A -85,B 0,C 180,E1 -8592.603,E2 -8592.603} C_VEL
LIN {X 0,Y 446.45,Z 528.864,A -85,B 0,C 180,E1 -8595.102,E2 -8595.102} C_VEL
LIN {X 0,Y 446.431,Z 528.872,A -85,B 0,C 180,E1 -8598.609,E2 -8598.609} C_VEL
LIN {X 0,Y 446.471,Z 528.86,A -85,B 0,C 180,E1 -8600.975,E2 -8600.975} C_VEL
LIN {X 0,Y 446.419,Z 528.873,A -85,B 0,C 180,E1 -8604.374,E2 -8604.374} C_VEL
LIN {X 0,Y 446.417,Z 528.876,A -85,B 0,C 180,E1 -8607.638,E2 -8607.638} C_VEL
LIN {X 0,Y 446.463,Z 528.868,A -85,B 0,C 180,E1 -8610.792,E2 -8610.792} C_VEL
LIN {X 0,Y 446.471,Z 528.87,A -85,B 0,C 180,E1 -8613.848,E2 -8613.848} C_VEL
LIN {X 0,Y 446.422,Z 528.872,A -85,B 0,C 180,E1 -8616.823,E2 -8616.823} C_VEL
LIN {X 0,Y 446.438,Z 528.875,A -85,B 0,C 180,E1 -8619.737,E2 -8619.737} C_VEL
LIN {X 0,Y 446.457,Z 528.865,A -85,B 0,C 180,E1 -8622.597,E2 -8622.597} C_VEL
LIN {X 0,Y 446.463,Z 528.869,A -85,B 0,C 180,E1 -8625.412,E2 -8625.412} C_VEL
LIN {X 0,Y 446.51,Z 528.86,A -85,B 0,C 180,E1 -8628.193,E2 -8628.193} C_VEL
LIN {X 0,Y 446.592,Z 528.855,A -85,B 0,C 180,E1 -8631.858,E2 -8631.858} C_VEL
